// TwinCAT 3 PLC project PLC1
// ProgramVersion: 3.1.4026.16
// CompilerDefines: VISU_USEPROPERTYINFO
// libraries:
//   SH_Light, * (StroemHansen)
//   Tc2_EnOcean, * (Beckhoff Automation GmbH)
//   Tc2_Standard, * (Beckhoff Automation GmbH)
//   Tc2_System, * (Beckhoff Automation GmbH)
//   Tc2_Utilities, * (Beckhoff Automation GmbH)
//   Tc3_DALI, * (Beckhoff Automation GmbH)
//   Tc3_System_DK, * (Beckhoff - DK)
//   VisuDialogs, * (System)
// project tree:
//   DUTs/DALI/ E_DALIExtendedFadeTime.TcTLEO (not stored), ST_DALI102Parameters.TcDUT (not stored), ST_DALI103Parameters.TcDUT (not stored), ST_DALIMemoryBank.TcDUT (not stored), ST_DALI_GrpAssignment.TcDUT (not stored), ST_GroupSort.TcDUT (not stored)
//   DUTs/EnOcean/ ST_ReadSAB05.TcDUT (not stored), ST_WriteSAB05.TcDUT (not stored)
//   / FastTask.TcTTO (not stored), GlobalTextList.TcGTLO (not stored), PlcTask.TcTTO (not stored), Visualization Manager.TcVMO (not stored)
//   GVLs/ GVL_AHDataModbus.TcGVL, GVL_EnOcean.TcGVL, GVL_Skalering.TcGVL (not stored)
//   POUs/01_System/01_System/GVLs/ GVL_EtherCAT.TcGVL (not stored)
//   POUs/01_System/01_System/ P_SystemDK.TcPOU (not stored)
//   POUs/AHModbusComm/ P_AHModbusComm.TcPOU
//   POUs/Alle_Rum/Gange/Gang_1_212A/ P_Gang_1_212A.TcPOU, Visualization_4_307_1_1_1_1.TcVIS (excluded from build)
//   POUs/Alle_Rum/Gange/Gang_1_216/ P_Gang_1_216.TcPOU, Visualization_4_308_1_2_1.TcVIS (excluded from build)
//   POUs/Alle_Rum/Gange/Gang_6_210/ P_Gang_6_210.TcPOU, Visualization_4_308_1_2_1_1.TcVIS (excluded from build)
//   POUs/Alle_Rum/Rum_Med_DALI_Pir/Rum_1_213/ P_Rum_1_213.TcPOU, Visualization_5_356_2_1_1_1.TcVIS (excluded from build)
//   POUs/Alle_Rum/Rum_Med_DALI_Pir/Rum_6_235/ P_Rum_6_235.TcPOU, Visualization_5_356_2_1_1_1_1.TcVIS (excluded from build)
//   POUs/Alle_Rum/Rum_Med_DALI_Pir/Rum_1_215/ P_Rum_1_215.TcPOU, Visualization_4_307_1_1_3_1_1_1.TcVIS (excluded from build)
//   POUs/Alle_Rum/Rum_Med_DALI_Pir/Rum_1_217/ P_Rum_1_217.TcPOU, Visualization_5_356_2_1_1_2.TcVIS (excluded from build)
//   POUs/Alle_Rum/Rum_Med_DALI_Pir/Rum_1_219/ P_Rum_1_219.TcPOU, Visualization_5_356_2_1_1_3.TcVIS (excluded from build)
//   POUs/Alle_Rum/Rum_Med_DALI_Pir/Rum_6_226B/ P_Rum_6_226B.TcPOU, Visualization_5_356_2_1_1_3_1.TcVIS (excluded from build)
//   POUs/Alle_Rum/Rum_Med_DALI_Pir/Rum_1_220/ P_Rum_1_220.TcPOU, Visualization_5_356_2_1_1_4.TcVIS (excluded from build)
//   POUs/Alle_Rum/Rum_Med_DALI_Pir/Rum_1_222/ P_Rum_1_222.TcPOU, Visualization_5_356_2_1_1_5.TcVIS (excluded from build)
//   POUs/Alle_Rum/Rum_Med_DALI_Pir/Rum_1_223/ P_Rum_1_223.TcPOU, Visualization_5_356_2_1_1_6.TcVIS (excluded from build)
//   POUs/Alle_Rum/Rum_Med_DALI_Pir/Rum_1_218/ P_Rum_1_218.TcPOU, Visualization_5_356_2_1_1.TcVIS (excluded from build)
//   POUs/Alle_Rum/Rum_Med_DALI_Pir/Rum_6_223/ P_Rum_6_223.TcPOU, Visualization_5_356_2_1_1_6_1.TcVIS (excluded from build)
//   POUs/Alle_Rum/Rum_Med_DALI_Pir/Rum_6_225/ P_Rum_6_225.TcPOU, Visualization_5_356_2_1_1_6_1_10.TcVIS (excluded from build)
//   POUs/Alle_Rum/Rum_Med_DALI_Pir/Rum_6_224/ P_Rum_6_224.TcPOU, Visualization_5_356_2_1_1_6_1_1.TcVIS (excluded from build)
//   POUs/Alle_Rum/Rum_Med_DALI_Pir/Rum_6_226A/ P_Rum_6_226A.TcPOU, Visualization_5_356_2_1_1_6_1_2.TcVIS (excluded from build)
//   POUs/Alle_Rum/Rum_Med_DALI_Pir/Rum_6_227/ P_Rum_6_227.TcPOU, Visualization_5_356_2_1_1_6_1_3.TcVIS (excluded from build)
//   POUs/Alle_Rum/Rum_Med_DALI_Pir/Rum_6_228/ P_Rum_6_228.TcPOU, Visualization_5_356_2_1_1_6_1_4.TcVIS (excluded from build)
//   POUs/Alle_Rum/Rum_Med_DALI_Pir/Rum_6_229/ P_Rum_6_229.TcPOU, Visualization_5_356_2_1_1_6_1_5.TcVIS (excluded from build)
//   POUs/Alle_Rum/Rum_Med_DALI_Pir/Rum_6_230/ P_Rum_6_230.TcPOU, Visualization_5_356_2_1_1_6_1_6.TcVIS (excluded from build)
//   POUs/Alle_Rum/Rum_Med_DALI_Pir/Rum_6_231/ P_Rum_6_231.TcPOU, Visualization_5_356_2_1_1_6_1_7.TcVIS (excluded from build)
//   POUs/Alle_Rum/Rum_Med_DALI_Pir/Rum_6_233/ P_Rum_6_233.TcPOU, Visualization_5_356_2_1_1_6_1_8.TcVIS (excluded from build)
//   POUs/Alle_Rum/Trapper/ P_Trappe.TcPOU (excluded from build)
//   POUs/DALI/DALI_Setup/ DALI_Commissioning.TcPOU (not stored)
//   POUs/DALI/DALI_Setup/FBs/ FB_Part102Addressing.TcPOU (not stored), FB_Part102Commands.TcPOU (not stored), FB_Part102Groups.TcPOU, FB_Part102MemoryPages.TcPOU (not stored), FB_Part102Parameters.TcPOU (not stored), FB_Part102Scenes.TcPOU (not stored), FB_Part102SetFading.TcPOU (not stored), FB_Part103Addressing.TcPOU (not stored), FB_Part103Identify.TcPOU (not stored), FB_Part103MemoryPages.TcPOU (not stored), FB_Part103Parameters.TcPOU (not stored), FB_Part202Emergency.TcPOU (not stored), FB_Part205Incandescent.TcPOU, FB_Part207LED.TcPOU, FB_Part208Switching.TcPOU (not stored), FB_Part300GenericDevice.TcPOU (not stored), FB_Part301PushButton.TcPOU (not stored), FB_Part302AbsoluteInputDevice.TcPOU (not stored), FB_Part303OccupancySensor.TcPOU (not stored), FB_Part304LightSensor.TcPOU (not stored), GearType.TcPOU (not stored)
//   POUs/DALI/DALI_Setup/GVLs/ GVL_Internal.TcGVL (not stored)
//   POUs/DALI/DALI_Setup/VISUs/TextLists/ CommandOnTerminalEvent.TcTLO, DimmingCurve.TcTLO (not stored), EventPriority.TcTLO (not stored), EventScheme.TcTLO, ExtendedFadeTime.TcTLO, FadeRate.TcTLO (not stored), FadeTime.TcTLO (not stored), FastFadeTime.TcTLO (not stored), TextList_Dialogs.TcTLO (not stored)
//   POUs/DALI/DALI_Setup/VISUs/ Visu_DALICommissioning.TcVIS
//   POUs/DALI/DALI_Setup/VISUs/Visu_DALICommissioning/ Visu_KL6821Configuration.TcVIS (not stored) (excluded from build), Visu_Part102Addressing.TcVIS, Visu_Part102Commands.TcVIS (not stored), Visu_Part102Groups.TcVIS (not stored), Visu_Part102MemoryBank.TcVIS (not stored), Visu_Part102Parameters.TcVIS, Visu_Part102Scenes.TcVIS, Visu_Part102SetFading.TcVIS (not stored), Visu_Part103Addressing.TcVIS (not stored), Visu_Part103Identify.TcVIS (not stored), Visu_Part103MemoryBank.TcVIS (not stored), Visu_Part103Parameters.TcVIS, Visu_Part202.TcVIS (not stored), Visu_Part202Commands.TcVIS, Visu_Part202Parameters.TcVIS, Visu_Part202Status.TcVIS (not stored), Visu_Part205.TcVIS (not stored), Visu_Part205Parameters.TcVIS (not stored), Visu_Part205Status.TcVIS (not stored), Visu_Part207.TcVIS (not stored), Visu_Part207Parameters.TcVIS (not stored), Visu_Part207Status.TcVIS (not stored), Visu_Part208Switching.TcVIS (not stored), Visu_Part300GenericDevice.TcVIS (not stored), Visu_Part301PushButton.TcVIS (not stored), Visu_Part302AbsoluteInputDevice.TcVIS (not stored), Visu_Part303OccupancySensor.TcVIS (not stored), Visu_Part304LightSensor.TcVIS (not stored), Visu_Welcome.TcVIS (not stored)
//   POUs/DALI/PRGs/Background/ P_DALI_Background.TcPOU (not stored)
//   POUs/DALI/PRGs/Diag/ P_DALI_DIAG.TcPOU (not stored)
//   POUs/DALI/PRGs/EnergyData/ P_DALI_Energy_Firmware_Test.TcPOU (not stored) (excluded from build), P_DALI_Energy_Line.TcPOU (not stored)
//   POUs/EnOcean/ P_EnOcean.TcPOU
//   POUs/ MAIN.TcPOU
// real-time tasks:
//   TASK PlcTask: cycle T#40ms, priority 21, ADS port 350
//   TASK FastTask: cycle T#4ms, priority 20, ADS port 351
// I/O:
//   DEVICE Device 1 (Beckhoff CCAT)
//   DEVICE Device 3 (CX-BK)
//     Box 1 (CX-BK)
// variable links:
//   PLC1/PLC1 Instance <-> Device 3 (CX-BK)/Box 1 (CX-BK)
//     FastTask Inputs/P_DALI_Background.arrKL6821InData[1] @bit 16 <-> Term 3 (KL6821)/Channel 1/Data In 0
//     FastTask Inputs/P_DALI_Background.arrKL6821InData[1] @bit 24 <-> Term 3 (KL6821)/Channel 1/Data In 1
//     FastTask Inputs/P_DALI_Background.arrKL6821InData[1] @bit 32 <-> Term 3 (KL6821)/Channel 1/Data In 2
//     FastTask Inputs/P_DALI_Background.arrKL6821InData[1] @bit 40 <-> Term 3 (KL6821)/Channel 1/Data In 3
//     FastTask Inputs/P_DALI_Background.arrKL6821InData[2] @bit 16 <-> Term 4 (KL6821)/Channel 1/Data In 0
//     FastTask Inputs/P_DALI_Background.arrKL6821InData[2] @bit 24 <-> Term 4 (KL6821)/Channel 1/Data In 1
//     FastTask Inputs/P_DALI_Background.arrKL6821InData[2] @bit 32 <-> Term 4 (KL6821)/Channel 1/Data In 2
//     FastTask Inputs/P_DALI_Background.arrKL6821InData[2] @bit 40 <-> Term 4 (KL6821)/Channel 1/Data In 3
//     FastTask Inputs/P_DALI_Background.arrKL6821InData[3] @bit 16 <-> Term 5 (KL6821)/Channel 1/Data In 0
//     FastTask Inputs/P_DALI_Background.arrKL6821InData[3] @bit 24 <-> Term 5 (KL6821)/Channel 1/Data In 1
//     FastTask Inputs/P_DALI_Background.arrKL6821InData[3] @bit 32 <-> Term 5 (KL6821)/Channel 1/Data In 2
//     FastTask Inputs/P_DALI_Background.arrKL6821InData[3] @bit 40 <-> Term 5 (KL6821)/Channel 1/Data In 3
//     FastTask Inputs/P_DALI_Background.arrKL6821InData[4] @bit 16 <-> Term 6 (KL6821)/Channel 1/Data In 0
//     FastTask Inputs/P_DALI_Background.arrKL6821InData[4] @bit 24 <-> Term 6 (KL6821)/Channel 1/Data In 1
//     FastTask Inputs/P_DALI_Background.arrKL6821InData[4] @bit 32 <-> Term 6 (KL6821)/Channel 1/Data In 2
//     FastTask Inputs/P_DALI_Background.arrKL6821InData[4] @bit 40 <-> Term 6 (KL6821)/Channel 1/Data In 3
//     FastTask Inputs/P_DALI_Background.arrKL6821InData[{1..4}] <-> Term {3..6} (KL6821)/Channel 1/State  (4 links)
//     FastTask Inputs/P_EnOcean.stKL6581_in @bit 8 <-> Term 2 (KL6581)/Channel 1/Input CNODE
//     FastTask Inputs/P_EnOcean.stKL6581_in @bit {24..48 step 8} <-> Term 2 (KL6581)/Channel 1/Input DB{0..3}  (4 links)
//     FastTask Inputs/P_EnOcean.stKL6581_in @bit {56..80 step 8} <-> Term 2 (KL6581)/Channel 1/Input ID{0..3}  (4 links)
//     FastTask Inputs/P_EnOcean.stKL6581_in @bit 16 <-> Term 2 (KL6581)/Channel 1/Input ORG
//     FastTask Inputs/P_EnOcean.stKL6581_in @bit 88 <-> Term 2 (KL6581)/Channel 1/Input STATUS
//     FastTask Inputs/P_EnOcean.stKL6581_in <-> Term 2 (KL6581)/Channel 1/Status
//     FastTask Outputs/P_DALI_Background.arrKL6821OutData[{1..4}] <-> Term {3..6} (KL6821)/Channel 1/Ctrl  (4 links)
//     FastTask Outputs/P_DALI_Background.arrKL6821OutData[1] @bit 16 <-> Term 3 (KL6821)/Channel 1/Data Out 0
//     FastTask Outputs/P_DALI_Background.arrKL6821OutData[1] @bit 24 <-> Term 3 (KL6821)/Channel 1/Data Out 1
//     FastTask Outputs/P_DALI_Background.arrKL6821OutData[1] @bit 32 <-> Term 3 (KL6821)/Channel 1/Data Out 2
//     FastTask Outputs/P_DALI_Background.arrKL6821OutData[1] @bit 40 <-> Term 3 (KL6821)/Channel 1/Data Out 3
//     FastTask Outputs/P_DALI_Background.arrKL6821OutData[2] @bit 16 <-> Term 4 (KL6821)/Channel 1/Data Out 0
//     FastTask Outputs/P_DALI_Background.arrKL6821OutData[2] @bit 24 <-> Term 4 (KL6821)/Channel 1/Data Out 1
//     FastTask Outputs/P_DALI_Background.arrKL6821OutData[2] @bit 32 <-> Term 4 (KL6821)/Channel 1/Data Out 2
//     FastTask Outputs/P_DALI_Background.arrKL6821OutData[2] @bit 40 <-> Term 4 (KL6821)/Channel 1/Data Out 3
//     FastTask Outputs/P_DALI_Background.arrKL6821OutData[3] @bit 16 <-> Term 5 (KL6821)/Channel 1/Data Out 0
//     FastTask Outputs/P_DALI_Background.arrKL6821OutData[3] @bit 24 <-> Term 5 (KL6821)/Channel 1/Data Out 1
//     FastTask Outputs/P_DALI_Background.arrKL6821OutData[3] @bit 32 <-> Term 5 (KL6821)/Channel 1/Data Out 2
//     FastTask Outputs/P_DALI_Background.arrKL6821OutData[3] @bit 40 <-> Term 5 (KL6821)/Channel 1/Data Out 3
//     FastTask Outputs/P_DALI_Background.arrKL6821OutData[4] @bit 16 <-> Term 6 (KL6821)/Channel 1/Data Out 0
//     FastTask Outputs/P_DALI_Background.arrKL6821OutData[4] @bit 24 <-> Term 6 (KL6821)/Channel 1/Data Out 1
//     FastTask Outputs/P_DALI_Background.arrKL6821OutData[4] @bit 32 <-> Term 6 (KL6821)/Channel 1/Data Out 2
//     FastTask Outputs/P_DALI_Background.arrKL6821OutData[4] @bit 40 <-> Term 6 (KL6821)/Channel 1/Data Out 3
//     FastTask Outputs/P_EnOcean.stKL6581_out <-> Term 2 (KL6581)/Channel 1/Control
//     FastTask Outputs/P_EnOcean.stKL6581_out @bit 8 <-> Term 2 (KL6581)/Channel 1/Output CNODE
//     FastTask Outputs/P_EnOcean.stKL6581_out @bit {24..48 step 8} <-> Term 2 (KL6581)/Channel 1/Output DB{0..3}  (4 links)
//     FastTask Outputs/P_EnOcean.stKL6581_out @bit {56..80 step 8} <-> Term 2 (KL6581)/Channel 1/Output ID{0..3}  (4 links)
//     FastTask Outputs/P_EnOcean.stKL6581_out @bit 16 <-> Term 2 (KL6581)/Channel 1/Output ORG
//     FastTask Outputs/P_EnOcean.stKL6581_out @bit 88 <-> Term 2 (KL6581)/Channel 1/Output STATUS
//     PlcTask Inputs/MAIN.nCX8200_State <-> Inputs/State

// ---- GVLs/GVL_AHDataModbus.TcGVL
{attribute 'qualified_only'}
{attribute 'qualified_only'}
VAR_GLOBAL
//AH pir data out
	nAH_NeighborRoomsPir_Out		AT %MB600	: UINT;
	
//AH pir data in
	arrAH_NeighborRoomsPir_In								: ARRAY[1..byNumberOfAH_Neighbors] OF UINT;
	arrAH_NeighborRoomsPir										: ARRAY[1..byNumberOfAH_Neighbors] OF ARRAY[0..15] OF BOOL;
	
//Schneider data out
	nCX8200_State_MB						AT %MB1000		: UINT;
	arrFB_DALIDiagErrorId		(*AT %MW1002*)		: ARRAY[1..SH_Light.DALI_Param.MAX_DALIV2_LINES] OF UDINT;
	arrKL6821InDataStatus					AT %MB1014		: ARRAY[1..SH_Light.DALI_Param.MAX_DALIV2_LINES] OF WORD;
	arrDALILineShrtAddrErr				AT %MB1026		: ARRAY[1..SH_Light.DALI_Param.MAX_DALIV2_LINES] OF UINT;
	EnOceanError								AT %MB1038		: UINT;
	nTotalEnergy10kWh						AT %MB1040		: UINT;
	nMaxControlGearOperatingHours	AT %MB1042		: UINT;
	uiPirOffDelayTimeAllRooms_MB   AT %MB1044   : UINT := 30;
END_VAR

VAR_GLOBAL CONSTANT
	byNumberOfAH_Neighbors									: BYTE := 25;
END_VAR


(*
AH2-2 pirsignaler = arrAH_NeighborRoomsPir[1]
	---------- KOPI fra A_AHNeighborRoomsPirOut i AH2-2 ----------
	GVL_AHDataModbus.nAH_NeighborRoomsPir_Out.0		:= P_Gang_2_244A.bPirActive_MB;
	GVL_AHDataModbus.nAH_NeighborRoomsPir_Out.1		:= P_Gang_7_201.bPirActive_MB;
*)

(*
AH6-2 pirsignaler = arrAH_NeighborRoomsPir[2]
	---------- KOPI fra A_AHNeighborRoomsPirOut i AH6-2 ----------
	
*)

// ---- GVLs/GVL_EnOcean.TcGVL
{attribute 'qualified_only'}
VAR_GLOBAL

//Gange
	strEnOceanSwitch_Gang_1_216_Pendler     			: Tc2_EnOcean.STR_EnOceanSwitch;

//Rum
	strEnOceanSwitch_Rum_1_213_Indgang				: Tc2_EnOcean.STR_EnOceanSwitch;
	strEnOceanSwitch_Rum_1_213_Ekstra					: Tc2_EnOcean.STR_EnOceanSwitch;
	
	strEnOceanSwitch_Rum_1_215								: Tc2_EnOcean.STR_EnOceanSwitch;
	strEnOceanSwitch_Rum_1_217								: Tc2_EnOcean.STR_EnOceanSwitch;
	strEnOceanSwitch_Rum_1_218								: Tc2_EnOcean.STR_EnOceanSwitch;
	strEnOceanSwitch_Rum_1_219								: Tc2_EnOcean.STR_EnOceanSwitch;
	strEnOceanSwitch_Rum_1_220								: Tc2_EnOcean.STR_EnOceanSwitch;
	strEnOceanSwitch_Rum_1_222								: Tc2_EnOcean.STR_EnOceanSwitch;
	strEnOceanSwitch_Rum_1_223								: Tc2_EnOcean.STR_EnOceanSwitch;
	
	strEnOceanSwitch_Rum_6_223								: Tc2_EnOcean.STR_EnOceanSwitch;
	strEnOceanSwitch_Rum_6_224								: Tc2_EnOcean.STR_EnOceanSwitch;
	strEnOceanSwitch_Rum_6_225								: Tc2_EnOcean.STR_EnOceanSwitch;
	strEnOceanSwitch_Rum_6_226A							: Tc2_EnOcean.STR_EnOceanSwitch;
	
	strEnOceanSwitch_Rum_6_226B_Indgang				: Tc2_EnOcean.STR_EnOceanSwitch;
	strEnOceanSwitch_Rum_6_226B_Pendler				: Tc2_EnOcean.STR_EnOceanSwitch;
	
	strEnOceanSwitch_Rum_6_227								: Tc2_EnOcean.STR_EnOceanSwitch;
	strEnOceanSwitch_Rum_6_228								: Tc2_EnOcean.STR_EnOceanSwitch;
	strEnOceanSwitch_Rum_6_229								: Tc2_EnOcean.STR_EnOceanSwitch;
	strEnOceanSwitch_Rum_6_230								: Tc2_EnOcean.STR_EnOceanSwitch;
	strEnOceanSwitch_Rum_6_231								: Tc2_EnOcean.STR_EnOceanSwitch;
	strEnOceanSwitch_Rum_6_233								: Tc2_EnOcean.STR_EnOceanSwitch;
	
	strEnOceanSwitch_Rum_6_235_Indgang				: Tc2_EnOcean.STR_EnOceanSwitch;
	strEnOceanSwitch_Rum_6_235_Ekstra					: Tc2_EnOcean.STR_EnOceanSwitch;
END_VAR

// ---- POUs/AHModbusComm/P_AHModbusComm.TcPOU
PROGRAM P_AHModbusComm
VAR
	arrfbReadAHPirData	: ARRAY[1..GVL_AHDataModbus.byNumberOfAH_Neighbors] OF SH_Light.FB_ReadAHPirData;
	arrReadAHPirData		: ARRAY[1..GVL_AHDataModbus.byNumberOfAH_Neighbors] OF BOOL;
	
	arrfbTriggerPulses			: ARRAY[1..GVL_AHDataModbus.byNumberOfAH_Neighbors] OF SH_Light.FB_ClockPulse;
	arrGeneratePulses			: ARRAY[1..GVL_AHDataModbus.byNumberOfAH_Neighbors] OF BOOL := [GVL_AHDataModbus.byNumberOfAH_Neighbors(TRUE)];
	tTimeInterval					: TIME := T#1S;
	tPulseTime					: TIME := T#1S;
	
	byLineId						: BYTE;
	byAHId						: BYTE;
	
		
	fbWritePirDelayTime		: R_TRIG;
	bRunOverrideOnce		: BOOL := FALSE;
	bEnableDelayTimeOverride : BOOL := FALSE;
	uiPirOffDelayTimeAllRooms : UINT := 30;
END_VAR

VAR CONSTANT
	arrnMBAddr					: ARRAY[1..GVL_AHDataModbus.byNumberOfAH_Neighbors] OF WORD := [GVL_AHDataModbus.byNumberOfAH_Neighbors(12588)]; //modbus-adresser (%MB600=>12588 default)
	arrstNeighborIPAddr		: ARRAY[1..GVL_AHDataModbus.byNumberOfAH_Neighbors] OF SH_Light.ST_NeighborIP := [
																						(sPLCName := 'AH1-1', sIP := '172.24.195.161', IsNeighbor := FALSE),
																						(sPLCName := 'AH1-2', sIP := '172.24.195.162', IsNeighbor := FALSE),	//Local must be false
																						(sPLCName := 'AH1-3', sIP := '172.24.195.163', IsNeighbor := FALSE),
																						(sPLCName := 'AH2-1', sIP := '172.24.195.164', IsNeighbor := FALSE),
																					(sPLCName := 'AH2-2', sIP := '172.24.195.165', IsNeighbor := TRUE),
																						(sPLCName := 'AH2-3', sIP := '172.24.195.166', IsNeighbor := FALSE),
																						(sPLCName := 'AH2-4', sIP := '172.24.195.167', IsNeighbor := FALSE),
																						(sPLCName := 'AH2-5', sIP := '172.24.195.168', IsNeighbor := FALSE),
																						(sPLCName := 'AH3-2', sIP := '172.24.195.169', IsNeighbor := FALSE),
																						(sPLCName := 'AH3-3', sIP := '172.24.195.170', IsNeighbor := FALSE),
																						(sPLCName := 'AH3-4', sIP := '172.24.195.171', IsNeighbor := FALSE),
																						(sPLCName := 'AH3-5', sIP := '172.24.195.172', IsNeighbor := FALSE),
																						(sPLCName := 'AH4-1', sIP := '172.24.195.173', IsNeighbor := FALSE),
																						(sPLCName := 'AH4-2', sIP := '172.24.195.174', IsNeighbor := FALSE),
																						(sPLCName := 'AH4-3', sIP := '172.24.195.175', IsNeighbor := FALSE),
																						(sPLCName := 'AH4-4', sIP := '172.24.195.176', IsNeighbor := FALSE),
																						(sPLCName := 'AH4-5', sIP := '172.24.195.177', IsNeighbor := FALSE),
																						(sPLCName := 'AH5-1', sIP := '172.24.195.178', IsNeighbor := FALSE),
																						(sPLCName := 'AH5-2', sIP := '172.24.195.179', IsNeighbor := FALSE),
																						(sPLCName := 'AH5-3', sIP := '172.24.195.180', IsNeighbor := FALSE),
																						(sPLCName := 'AH5-4', sIP := '172.24.195.181', IsNeighbor := FALSE),
																						(sPLCName := 'AH5-5', sIP := '172.24.195.182', IsNeighbor := FALSE),
																						(sPLCName := 'AH6-1', sIP := '172.24.195.183', IsNeighbor := FALSE),
																					(sPLCName := 'AH6-2', sIP := '172.24.195.184', IsNeighbor := TRUE),
																						(sPLCName := 'AH6-3', sIP := '172.24.195.185', IsNeighbor := FALSE)];
																					//	(sPLCName := 'AH3-1', sIP := '172.24.195.186', IsNeighbor := TRUE) //when ready
END_VAR

A_AHNeighborRoomsPirIn();
A_AHNeighborRoomsPirOut();
A_DALILineShrtAddrErr();
A_DelayTimeAllRooms();

ACTION A_AHNeighborRoomsPirIn:
FOR byAHId := 1 TO GVL_AHDataModbus.byNumberOfAH_Neighbors DO
	IF arrstNeighborIPAddr[byAHId].IsNeighbor THEN
		//Generate Pulses
		arrfbTriggerPulses[byAHId](bGenerateClockPulses:= arrGeneratePulses[byAHId], tTimeInterval:= tTimeInterval, tPulseTime:= tPulseTime);
		arrReadAHPirData[byAHId]:= arrfbTriggerPulses[byAHId].bPulse;
		//Read data
		arrfbReadAHPirData[byAHId](	bReadAHPirData				:=	arrReadAHPirData[byAHId],
														sIPAddr							:=	arrstNeighborIPAddr[byAHId].sIP,
														nMBAddr							:=	arrnMBAddr[byAHId],
														nMBDataBuffer				:=	GVL_AHDataModbus.arrAH_NeighborRoomsPir_In[byAHId],
														arrAH_NeighborRoomsPir	=>GVL_AHDataModbus.arrAH_NeighborRoomsPir[byAHId]);
	END_IF
END_FOR
END_ACTION

ACTION A_AHNeighborRoomsPirOut:
GVL_AHDataModbus.nAH_NeighborRoomsPir_Out.0 := P_Gang_1_216.bPirActive_MB;
GVL_AHDataModbus.nAH_NeighborRoomsPir_Out.1 := P_Gang_6_210.bPirActive_MB;
//GVL_AHDataModbus.nAH_NeighborRoomsPir_Out.2 :=
//GVL_AHDataModbus.nAH_NeighborRoomsPir_Out.3 := 
//GVL_AHDataModbus.nAH_NeighborRoomsPir_Out.4 :=
//GVL_AHDataModbus.nAH_NeighborRoomsPir_Out.5 := 
//GVL_AHDataModbus.nAH_NeighborRoomsPir_Out.6 :=
//GVL_AHDataModbus.nAH_NeighborRoomsPir_Out.7 := 
//GVL_AHDataModbus.nAH_NeighborRoomsPir_Out.8 :=
//GVL_AHDataModbus.nAH_NeighborRoomsPir_Out.9 := 
//GVL_AHDataModbus.nAH_NeighborRoomsPir_Out.10 :=
//GVL_AHDataModbus.nAH_NeighborRoomsPir_Out.11 := 
//GVL_AHDataModbus.nAH_NeighborRoomsPir_Out.12 := 
//GVL_AHDataModbus.nAH_NeighborRoomsPir_Out.13 := 
//GVL_AHDataModbus.nAH_NeighborRoomsPir_Out.14 := 
//GVL_AHDataModbus.nAH_NeighborRoomsPir_Out.15 :=
END_ACTION

ACTION A_DALILineShrtAddrErr:
FOR  byLineId := 1 TO SH_Light.DALI_Param.MAX_DALIV2_LINES DO
	GVL_AHDataModbus.arrDALILineShrtAddrErr[byLineId] :=  TO_UINT(SH_Light.GVL_DALI_LatestError.arrLineShrtAddr[byLineId]);
END_FOR
END_ACTION

ACTION A_DelayTimeAllRooms:

fbWritePirDelayTime(CLK := GVL_AHDataModbus.uiPirOffDelayTimeAllRooms_MB<>uiPirOffDelayTimeAllRooms);

IF fbWritePirDelayTime.Q THEN
	bRunOverrideOnce := TRUE;
	bEnableDelayTimeOverride := TRUE;
	
//Indsæt kode
P_Gang_1_212A.fbWritePirDelayTIme(bEnableOverride := bEnableDelayTimeOverride, nOverRideValue := GVL_AHDataModbus.uiPirOffDelayTimeAllRooms_MB, nValIn1 := GVL_AHDataModbus.uiPirOffDelayTimeAllRooms_MB, nValIn2 := uiPirOffDelayTimeAllRooms);
P_Gang_1_216.fbWritePirDelayTIme(bEnableOverride := bEnableDelayTimeOverride, nOverRideValue := GVL_AHDataModbus.uiPirOffDelayTimeAllRooms_MB, nValIn1 := GVL_AHDataModbus.uiPirOffDelayTimeAllRooms_MB, nValIn2 := uiPirOffDelayTimeAllRooms);
P_Gang_6_210.fbWritePirDelayTIme(bEnableOverride := bEnableDelayTimeOverride, nOverRideValue := GVL_AHDataModbus.uiPirOffDelayTimeAllRooms_MB, nValIn1 := GVL_AHDataModbus.uiPirOffDelayTimeAllRooms_MB, nValIn2 := uiPirOffDelayTimeAllRooms);
P_Rum_1_213.fbWritePirDelayTIme(bEnableOverride := bEnableDelayTimeOverride, nOverRideValue := GVL_AHDataModbus.uiPirOffDelayTimeAllRooms_MB, nValIn1 := GVL_AHDataModbus.uiPirOffDelayTimeAllRooms_MB, nValIn2 := uiPirOffDelayTimeAllRooms);
P_Rum_1_215.fbWritePirDelayTIme(bEnableOverride := bEnableDelayTimeOverride, nOverRideValue := GVL_AHDataModbus.uiPirOffDelayTimeAllRooms_MB, nValIn1 := GVL_AHDataModbus.uiPirOffDelayTimeAllRooms_MB, nValIn2 := uiPirOffDelayTimeAllRooms);
P_Rum_1_217.fbWritePirDelayTIme(bEnableOverride := bEnableDelayTimeOverride, nOverRideValue := GVL_AHDataModbus.uiPirOffDelayTimeAllRooms_MB, nValIn1 := GVL_AHDataModbus.uiPirOffDelayTimeAllRooms_MB, nValIn2 := uiPirOffDelayTimeAllRooms);
P_Rum_1_218.fbWritePirDelayTIme(bEnableOverride := bEnableDelayTimeOverride, nOverRideValue := GVL_AHDataModbus.uiPirOffDelayTimeAllRooms_MB, nValIn1 := GVL_AHDataModbus.uiPirOffDelayTimeAllRooms_MB, nValIn2 := uiPirOffDelayTimeAllRooms);
P_Rum_1_219.fbWritePirDelayTIme(bEnableOverride := bEnableDelayTimeOverride, nOverRideValue := GVL_AHDataModbus.uiPirOffDelayTimeAllRooms_MB, nValIn1 := GVL_AHDataModbus.uiPirOffDelayTimeAllRooms_MB, nValIn2 := uiPirOffDelayTimeAllRooms);
P_Rum_1_222.fbWritePirDelayTIme(bEnableOverride := bEnableDelayTimeOverride, nOverRideValue := GVL_AHDataModbus.uiPirOffDelayTimeAllRooms_MB, nValIn1 := GVL_AHDataModbus.uiPirOffDelayTimeAllRooms_MB, nValIn2 := uiPirOffDelayTimeAllRooms);
P_Rum_1_220.fbWritePirDelayTIme(bEnableOverride := bEnableDelayTimeOverride, nOverRideValue := GVL_AHDataModbus.uiPirOffDelayTimeAllRooms_MB, nValIn1 := GVL_AHDataModbus.uiPirOffDelayTimeAllRooms_MB, nValIn2 := uiPirOffDelayTimeAllRooms);
P_Rum_1_223.fbWritePirDelayTIme(bEnableOverride := bEnableDelayTimeOverride, nOverRideValue := GVL_AHDataModbus.uiPirOffDelayTimeAllRooms_MB, nValIn1 := GVL_AHDataModbus.uiPirOffDelayTimeAllRooms_MB, nValIn2 := uiPirOffDelayTimeAllRooms);
P_Rum_6_223.fbWritePirDelayTIme(bEnableOverride := bEnableDelayTimeOverride, nOverRideValue := GVL_AHDataModbus.uiPirOffDelayTimeAllRooms_MB, nValIn1 := GVL_AHDataModbus.uiPirOffDelayTimeAllRooms_MB, nValIn2 := uiPirOffDelayTimeAllRooms);
P_Rum_6_224.fbWritePirDelayTIme(bEnableOverride := bEnableDelayTimeOverride, nOverRideValue := GVL_AHDataModbus.uiPirOffDelayTimeAllRooms_MB, nValIn1 := GVL_AHDataModbus.uiPirOffDelayTimeAllRooms_MB, nValIn2 := uiPirOffDelayTimeAllRooms);
P_Rum_6_225.fbWritePirDelayTIme(bEnableOverride := bEnableDelayTimeOverride, nOverRideValue := GVL_AHDataModbus.uiPirOffDelayTimeAllRooms_MB, nValIn1 := GVL_AHDataModbus.uiPirOffDelayTimeAllRooms_MB, nValIn2 := uiPirOffDelayTimeAllRooms);
P_Rum_6_226A.fbWritePirDelayTIme(bEnableOverride := bEnableDelayTimeOverride, nOverRideValue := GVL_AHDataModbus.uiPirOffDelayTimeAllRooms_MB, nValIn1 := GVL_AHDataModbus.uiPirOffDelayTimeAllRooms_MB, nValIn2 := uiPirOffDelayTimeAllRooms);
P_Rum_6_226B.fbWritePirDelayTIme(bEnableOverride := bEnableDelayTimeOverride, nOverRideValue := GVL_AHDataModbus.uiPirOffDelayTimeAllRooms_MB, nValIn1 := GVL_AHDataModbus.uiPirOffDelayTimeAllRooms_MB, nValIn2 := uiPirOffDelayTimeAllRooms);
P_Rum_6_227.fbWritePirDelayTIme(bEnableOverride := bEnableDelayTimeOverride, nOverRideValue := GVL_AHDataModbus.uiPirOffDelayTimeAllRooms_MB, nValIn1 := GVL_AHDataModbus.uiPirOffDelayTimeAllRooms_MB, nValIn2 := uiPirOffDelayTimeAllRooms);
P_Rum_6_228.fbWritePirDelayTIme(bEnableOverride := bEnableDelayTimeOverride, nOverRideValue := GVL_AHDataModbus.uiPirOffDelayTimeAllRooms_MB, nValIn1 := GVL_AHDataModbus.uiPirOffDelayTimeAllRooms_MB, nValIn2 := uiPirOffDelayTimeAllRooms);
P_Rum_6_229.fbWritePirDelayTIme(bEnableOverride := bEnableDelayTimeOverride, nOverRideValue := GVL_AHDataModbus.uiPirOffDelayTimeAllRooms_MB, nValIn1 := GVL_AHDataModbus.uiPirOffDelayTimeAllRooms_MB, nValIn2 := uiPirOffDelayTimeAllRooms);
P_Rum_6_230.fbWritePirDelayTIme(bEnableOverride := bEnableDelayTimeOverride, nOverRideValue := GVL_AHDataModbus.uiPirOffDelayTimeAllRooms_MB, nValIn1 := GVL_AHDataModbus.uiPirOffDelayTimeAllRooms_MB, nValIn2 := uiPirOffDelayTimeAllRooms);
P_Rum_6_231.fbWritePirDelayTIme(bEnableOverride := bEnableDelayTimeOverride, nOverRideValue := GVL_AHDataModbus.uiPirOffDelayTimeAllRooms_MB, nValIn1 := GVL_AHDataModbus.uiPirOffDelayTimeAllRooms_MB, nValIn2 := uiPirOffDelayTimeAllRooms);
P_Rum_6_233.fbWritePirDelayTIme(bEnableOverride := bEnableDelayTimeOverride, nOverRideValue := GVL_AHDataModbus.uiPirOffDelayTimeAllRooms_MB, nValIn1 := GVL_AHDataModbus.uiPirOffDelayTimeAllRooms_MB, nValIn2 := uiPirOffDelayTimeAllRooms);
P_Rum_6_235.fbWritePirDelayTIme(bEnableOverride := bEnableDelayTimeOverride, nOverRideValue := GVL_AHDataModbus.uiPirOffDelayTimeAllRooms_MB, nValIn1 := GVL_AHDataModbus.uiPirOffDelayTimeAllRooms_MB, nValIn2 := uiPirOffDelayTimeAllRooms);

ELSE
	IF bRunOverrideOnce THEN
		bEnableDelayTimeOverride := FALSE;
		
		//Indsæt kode
P_Gang_1_212A.fbWritePirDelayTIme(bEnableOverride := bEnableDelayTimeOverride, nOverRideValue := GVL_AHDataModbus.uiPirOffDelayTimeAllRooms_MB, nValIn1 := GVL_AHDataModbus.uiPirOffDelayTimeAllRooms_MB, nValIn2 := uiPirOffDelayTimeAllRooms);
P_Gang_1_216.fbWritePirDelayTIme(bEnableOverride := bEnableDelayTimeOverride, nOverRideValue := GVL_AHDataModbus.uiPirOffDelayTimeAllRooms_MB, nValIn1 := GVL_AHDataModbus.uiPirOffDelayTimeAllRooms_MB, nValIn2 := uiPirOffDelayTimeAllRooms);
P_Gang_6_210.fbWritePirDelayTIme(bEnableOverride := bEnableDelayTimeOverride, nOverRideValue := GVL_AHDataModbus.uiPirOffDelayTimeAllRooms_MB, nValIn1 := GVL_AHDataModbus.uiPirOffDelayTimeAllRooms_MB, nValIn2 := uiPirOffDelayTimeAllRooms);
P_Rum_1_213.fbWritePirDelayTIme(bEnableOverride := bEnableDelayTimeOverride, nOverRideValue := GVL_AHDataModbus.uiPirOffDelayTimeAllRooms_MB, nValIn1 := GVL_AHDataModbus.uiPirOffDelayTimeAllRooms_MB, nValIn2 := uiPirOffDelayTimeAllRooms);
P_Rum_1_215.fbWritePirDelayTIme(bEnableOverride := bEnableDelayTimeOverride, nOverRideValue := GVL_AHDataModbus.uiPirOffDelayTimeAllRooms_MB, nValIn1 := GVL_AHDataModbus.uiPirOffDelayTimeAllRooms_MB, nValIn2 := uiPirOffDelayTimeAllRooms);
P_Rum_1_217.fbWritePirDelayTIme(bEnableOverride := bEnableDelayTimeOverride, nOverRideValue := GVL_AHDataModbus.uiPirOffDelayTimeAllRooms_MB, nValIn1 := GVL_AHDataModbus.uiPirOffDelayTimeAllRooms_MB, nValIn2 := uiPirOffDelayTimeAllRooms);
P_Rum_1_218.fbWritePirDelayTIme(bEnableOverride := bEnableDelayTimeOverride, nOverRideValue := GVL_AHDataModbus.uiPirOffDelayTimeAllRooms_MB, nValIn1 := GVL_AHDataModbus.uiPirOffDelayTimeAllRooms_MB, nValIn2 := uiPirOffDelayTimeAllRooms);
P_Rum_1_219.fbWritePirDelayTIme(bEnableOverride := bEnableDelayTimeOverride, nOverRideValue := GVL_AHDataModbus.uiPirOffDelayTimeAllRooms_MB, nValIn1 := GVL_AHDataModbus.uiPirOffDelayTimeAllRooms_MB, nValIn2 := uiPirOffDelayTimeAllRooms);
P_Rum_1_222.fbWritePirDelayTIme(bEnableOverride := bEnableDelayTimeOverride, nOverRideValue := GVL_AHDataModbus.uiPirOffDelayTimeAllRooms_MB, nValIn1 := GVL_AHDataModbus.uiPirOffDelayTimeAllRooms_MB, nValIn2 := uiPirOffDelayTimeAllRooms);
P_Rum_1_220.fbWritePirDelayTIme(bEnableOverride := bEnableDelayTimeOverride, nOverRideValue := GVL_AHDataModbus.uiPirOffDelayTimeAllRooms_MB, nValIn1 := GVL_AHDataModbus.uiPirOffDelayTimeAllRooms_MB, nValIn2 := uiPirOffDelayTimeAllRooms);
P_Rum_1_223.fbWritePirDelayTIme(bEnableOverride := bEnableDelayTimeOverride, nOverRideValue := GVL_AHDataModbus.uiPirOffDelayTimeAllRooms_MB, nValIn1 := GVL_AHDataModbus.uiPirOffDelayTimeAllRooms_MB, nValIn2 := uiPirOffDelayTimeAllRooms);
P_Rum_6_223.fbWritePirDelayTIme(bEnableOverride := bEnableDelayTimeOverride, nOverRideValue := GVL_AHDataModbus.uiPirOffDelayTimeAllRooms_MB, nValIn1 := GVL_AHDataModbus.uiPirOffDelayTimeAllRooms_MB, nValIn2 := uiPirOffDelayTimeAllRooms);
P_Rum_6_224.fbWritePirDelayTIme(bEnableOverride := bEnableDelayTimeOverride, nOverRideValue := GVL_AHDataModbus.uiPirOffDelayTimeAllRooms_MB, nValIn1 := GVL_AHDataModbus.uiPirOffDelayTimeAllRooms_MB, nValIn2 := uiPirOffDelayTimeAllRooms);
P_Rum_6_225.fbWritePirDelayTIme(bEnableOverride := bEnableDelayTimeOverride, nOverRideValue := GVL_AHDataModbus.uiPirOffDelayTimeAllRooms_MB, nValIn1 := GVL_AHDataModbus.uiPirOffDelayTimeAllRooms_MB, nValIn2 := uiPirOffDelayTimeAllRooms);
P_Rum_6_226A.fbWritePirDelayTIme(bEnableOverride := bEnableDelayTimeOverride, nOverRideValue := GVL_AHDataModbus.uiPirOffDelayTimeAllRooms_MB, nValIn1 := GVL_AHDataModbus.uiPirOffDelayTimeAllRooms_MB, nValIn2 := uiPirOffDelayTimeAllRooms);
P_Rum_6_226B.fbWritePirDelayTIme(bEnableOverride := bEnableDelayTimeOverride, nOverRideValue := GVL_AHDataModbus.uiPirOffDelayTimeAllRooms_MB, nValIn1 := GVL_AHDataModbus.uiPirOffDelayTimeAllRooms_MB, nValIn2 := uiPirOffDelayTimeAllRooms);
P_Rum_6_227.fbWritePirDelayTIme(bEnableOverride := bEnableDelayTimeOverride, nOverRideValue := GVL_AHDataModbus.uiPirOffDelayTimeAllRooms_MB, nValIn1 := GVL_AHDataModbus.uiPirOffDelayTimeAllRooms_MB, nValIn2 := uiPirOffDelayTimeAllRooms);
P_Rum_6_228.fbWritePirDelayTIme(bEnableOverride := bEnableDelayTimeOverride, nOverRideValue := GVL_AHDataModbus.uiPirOffDelayTimeAllRooms_MB, nValIn1 := GVL_AHDataModbus.uiPirOffDelayTimeAllRooms_MB, nValIn2 := uiPirOffDelayTimeAllRooms);
P_Rum_6_229.fbWritePirDelayTIme(bEnableOverride := bEnableDelayTimeOverride, nOverRideValue := GVL_AHDataModbus.uiPirOffDelayTimeAllRooms_MB, nValIn1 := GVL_AHDataModbus.uiPirOffDelayTimeAllRooms_MB, nValIn2 := uiPirOffDelayTimeAllRooms);
P_Rum_6_230.fbWritePirDelayTIme(bEnableOverride := bEnableDelayTimeOverride, nOverRideValue := GVL_AHDataModbus.uiPirOffDelayTimeAllRooms_MB, nValIn1 := GVL_AHDataModbus.uiPirOffDelayTimeAllRooms_MB, nValIn2 := uiPirOffDelayTimeAllRooms);
P_Rum_6_231.fbWritePirDelayTIme(bEnableOverride := bEnableDelayTimeOverride, nOverRideValue := GVL_AHDataModbus.uiPirOffDelayTimeAllRooms_MB, nValIn1 := GVL_AHDataModbus.uiPirOffDelayTimeAllRooms_MB, nValIn2 := uiPirOffDelayTimeAllRooms);
P_Rum_6_233.fbWritePirDelayTIme(bEnableOverride := bEnableDelayTimeOverride, nOverRideValue := GVL_AHDataModbus.uiPirOffDelayTimeAllRooms_MB, nValIn1 := GVL_AHDataModbus.uiPirOffDelayTimeAllRooms_MB, nValIn2 := uiPirOffDelayTimeAllRooms);
P_Rum_6_235.fbWritePirDelayTIme(bEnableOverride := bEnableDelayTimeOverride, nOverRideValue := GVL_AHDataModbus.uiPirOffDelayTimeAllRooms_MB, nValIn1 := GVL_AHDataModbus.uiPirOffDelayTimeAllRooms_MB, nValIn2 := uiPirOffDelayTimeAllRooms);

		bRunOverrideOnce := FALSE;
	END_IF
END_IF
END_ACTION

END_PROGRAM

// ---- POUs/Alle_Rum/Gange/Gang_1_216/P_Gang_1_216.TcPOU
PROGRAM P_Gang_1_216
(*
Gangen består af en lysgruppe og et ekstra armatur - L2G2 og L1S38 - på to forskellige linjer
både gruppe og ekstra armatur afhænger af samme PIR-input : pir-adr. 5, 6 og 10 på DALI-linje 2 og pir-adr. 4 på DALI-linje 4
Derfor oprettes to adskilte reguleringer med samme PV. Dvs., at knapfunktion og pirfunktion forbliver den samme.
Der oprettes to sensor setups, som samles i A_Sensor.
Gangen nabostyres af Gang_1_216 fra AH2-2 og udvalgte rum på gangen
*)
VAR
	arrfbLysGruppe			: ARRAY [1..2] OF FB_Light_Type_B;
	arrstDaliSetupGruppe	: ARRAY[1..2] OF SH_Light.ST_DALI_RoomSetup := 
	
													[(	byShrtAdr_Prim	:= 11, 
														byGrpAdr_Prim		:= 2, 
														eMod_Prim			:= E_DALIAddressType.Group, 
														//byShrtAdr_Sec		:= 1, 
														//byGrpAdr_Sec		:= 1, 
														//eMod_Sec			:= E_DALIAddressType.Short, 
														byShrtAdr_Supl		:= 26,
														//byGrpAdr_Supl := 1,
														eMod_Supl			:= E_DALIAddressType.Short,
														DALI_LINE_NUM_PRIM	:= arrDALI_LINE_NUM_LIGHT[1], 
														DALI_LINE_NUM_SEC		:= 0, //0 = ingen zonestyring/vinduerække
														DALI_LINE_NUM_SUPL	:= arrDALI_LINE_NUM_PENDANTS[1]),
														
													(	byShrtAdr_Prim	:= 38, 
														byGrpAdr_Prim		:= 1, 
														eMod_Prim			:= E_DALIAddressType.Short, 
														//byShrtAdr_Sec		:= 1, 
														//byGrpAdr_Sec		:= 1, 
														//eMod_Sec			:= E_DALIAddressType.Short, 
														//byShrtAdr_Supl		:= 1,
														//byGrpAdr_Supl := 1,
														//eMod_Supl			:= E_DALIAddressType.Short, 
														DALI_LINE_NUM_PRIM	:= arrDALI_LINE_NUM_LIGHT[2], 
														DALI_LINE_NUM_SEC		:= 0, 
														DALI_LINE_NUM_SUPL	:= arrDALI_LINE_NUM_PENDANTS[2])];
	
	arrstLiveDataGruppe			: ARRAY [1..2] OF SH_Light.ST_LiveData;
	arrRunTuningGruppe			: ARRAY[1..2] OF BOOL;
	
	bTopButtonZone1				: BOOL;
	bTopButtonZone1_Visu		: BOOL;
	bBottomButtonZone1			: BOOL;
	bBottomButtonZone1_Visu	: BOOL;
	bButtonZone2					: BOOL;
	bNeighborRoomsPir			: BOOL;
	fLuxOn								: REAL;
	fLuxDim							: REAL;
	tPIRDim							: TIME;
	tPIROff							: TIME;
	fOffsetSec						: REAL := 20;
	bOccupiedRoom				: BOOL;

// Sensor Settings
	fbSensor						: SH_Light.FB_NIKO_P46xx_3Pcs;
	arrSensorAddr				: ARRAY[1..3] OF BYTE :=[5,6,10];  
	bInitialize						: BOOL := TRUE;
	stDaliSensorSetup			: ST_DALI_NIKOP46SetupData;
	arrInitErr						: ARRAY [1..3] OF BOOL;
	arrInitDone					: ARRAY [1..3] OF BOOL;
	arrSensorScales				: ARRAY [1..10] OF SH_Light.ST_DALI_SensorScaleMode := [
																							(fMeassureMaxSensor := rMeassure_Zone10, fReadMaxSensor := rRead_Zone10),
																							(fMeassureMaxSensor := rMeassure_Zone10, fReadMaxSensor := rRead_Zone10),
																							(fMeassureMaxSensor := rMeassure_Zone10, fReadMaxSensor := rRead_Zone10),
																							7(())];
	
	//Setup af sensorer på forskellige linjer kan ikke håndteres med ARRAYS som sædvanlig, da der kun er 1 sensor på setup 2.
	fbSensor2						: SH_Light.FB_NIKO_P46xx_1Pcs;
	bySensor2Addr				: BYTE := 4;
	bInitialize2						: BOOL := TRUE;
	stDaliSensor2Setup		: ST_DALI_NIKOP46SetupData;
	bInitErr2						: BOOL;
	bInitDone2					: BOOL;
	arrSensor2Scales			: ARRAY [1..10] OF SH_Light.ST_DALI_SensorScaleMode := [
																							(fMeassureMaxSensor := 1023, fReadMaxSensor := 1023),
																							9(())];
																					
	bCancelHoldTimerOccupancy	: BOOL;
	
(*	eEventPriorityOccupancy		: E_DALIEventPriority := E_DALIEVENTPRIORITY.Middle;
	nHoldTimerOccupancy			: WORD := 5; // Value in s. 	
	nReportTimerOccupancy		: BYTE := 120; // Value in s, Preset manufacturer value
	nDeadtimeTimerOccupancy		: WORD := 100; // Value in ms, Predefined Value of DALI Standard
	bCancelHoldTimerOccupancy	: BOOL;
	nSensitivityOccupancy		: BYTE:= 3; //setting Sensivity (0..4) 0 (Off), 1 (Min), 2(Low), 3(High) and 4 (Max)

	bEnableLuxEvent				: BOOL;
	eEventPriorityBrightness	: E_DALIEventPriority := E_DALIEVENTPRIORITY.Middle;
	nDeadtimeTimerBrightness	: WORD := 1500; // Value in ms, Predefined Value of DALI Standard
	nHysteresisBrightness		: BYTE := 2; // Value in %
	nHysteresisMinBrightness	: BYTE := 10; // Absolute Value, depending on the manufacturer specific resolution
	nReportTimerBrightness		: BYTE := 120; // Value in s, Preset manufacturer value
*)

	//ModbusComm setup
	
	fbWriteSPLuxLevel				: SH_Light.FB_TwoVal_SelectOne_RTrigChange;
	fbWritePirDelayTIme			: SH_Light.FB_TwoVal_SelectOne_RTrigChange;
	stRoomDataPLC					: SH_Light.ST_RoomDataPLC	:=	(
																		uiPirOffDelayTime	:= 30,
																		uiSpLuxLevel			:= 500,
																		uiPirDimDelayTime	:= 15,
																		uiSpDimLuxLevel		:= 200);
																		
	fbBallastOnHours				: SH_Light.FB_CountOnHours;
	bEnableHourCount			: BOOL := TRUE;
	
	//Non-persistent modbus data
	bPirActive_MB					AT %MX32.0	: BOOL;				//bPirLys i gammel kode
	uiActLuxLevel_MB			AT %MB36		: UINT;				//intHMIAktueltLux i gammel kode
	uiActLightLevelPct_MB	AT %MB40		: UINT;				//intDALI_Gruppe1_Lysniveau i gammel kode
	
	//For Conversion
	uiPirOffMinutes						: UINT;
	udTimeScaling						: UDINT := 60000;
	uiLuxOn								: UINT;
	
	//max values checks
	uiMaxLuxLevel						: UINT := 1023;
	uiMaxPirOffMinutes				: UINT := 180;

END_VAR

VAR CONSTANT
	Sensor_DALI_LINE_NUM		: BYTE := 2;
	Sensor2_DALI_LINE_NUM	: BYTE := 4;
    arrDALI_LINE_NUM_LIGHT: ARRAY[1..2] OF BYTE := [2,1]; //korrekt rækkefølge nødvendig //rækkefølge og linje 
	arrDALI_LINE_NUM_PENDANTS: ARRAY[1..2] OF BYTE := [2,0]; //korrekt rækkefølge nødvendig. 0 = ingen pendler
END_VAR
VAR PERSISTENT
	stPirSensorData			: SH_Light.ST_DALI_Sensor;
	arrstPirSensorDataLine	: ARRAY[1..2] OF SH_Light.ST_DALI_Sensor;
	arrstTuneDataGruppe	: ARRAY [1..2] OF SH_Light.ST_TuneData_EX;
	
	uiPirOffDelayTime_MB		AT %MB34	: UINT;				//ntHMI_Pir_SetValue i gammel kode
	uiSPLuxLevel_MB			AT %MB38	: UINT;				//intHMI_Lux_SetValue i gammel kode
	uiBallastOnHours_MB		AT %MB42	: UINT;				//dintHMILysbraendtimer1 i gammel kode
	byOnHoursOverflowCount						: BYTE;
END_VAR

A_Buttons();
A_LightCtrl();
A_ModbusComm();
A_Sensor();

ACTION A_Buttons:
bTopButtonZone1		:= bTopButtonZone1_Visu;
bBottomButtonZone1	:= bBottomButtonZone1_Visu;

bButtonZone2	:= GVL_EnOcean.strEnOceanSwitch_Gang_1_216_Pendler.bT2_OFF OR GVL_EnOcean.strEnOceanSwitch_Gang_1_216_Pendler.bT2_ON;
END_ACTION

ACTION A_LightCtrl:
bNeighborRoomsPir := 	P_Gang_1_212A.stPirSensorData.bPrc OR
									P_Rum_1_213.stPirSensorData.bPrc OR
									P_Rum_1_215.stPirSensorData.bPrc OR
									P_Rum_1_217.stPirSensorData.bPrc OR
									P_Rum_1_218.stPirSensorData.bPrc OR
									P_Rum_1_219.stPirSensorData.bPrc OR
									P_Rum_1_220.stPirSensorData.bPrc OR
									P_Rum_1_222.stPirSensorData.bPrc OR
									P_Rum_1_223.stPirSensorData.bPrc OR
									GVL_AHDataModbus.arrAH_NeighborRoomsPir[5][2] OR
									GVL_AHDataModbus.arrAH_NeighborRoomsPir[5][3] OR
									GVL_AHDataModbus.arrAH_NeighborRoomsPir[5][4] OR
									GVL_AHDataModbus.arrAH_NeighborRoomsPir[5][5];

arrfbLysGruppe[1]( 
	nZoneID:= 1, 
	bButtonZone1:= bTopButtonZone1,
	bBottomButtonZone1 := bBottomButtonZone1, 
	//bTopButtonOverride := ,
	//bBottomButtonOverride := ,
	bButtonZone2:= bButtonZone2,
	//bNoButtons := ,
	bNeighborRoomsPir	:=	bNeighborRoomsPir,
	fLuxOn:= fLuxOn, 
	fLuxDim:= fLuxDim, 
	tPIRDim:= tPIRDim, 
	tPIROff:= tPIROff, 
	fOffsetSec:= fOffsetSec, 
	bReInit:= , 
	stDaliSetup:= arrstDaliSetupGruppe[1], 
	ipCommunication_Prim:= P_DALI_Background.arrfbKL6821Communication[arrDALI_LINE_NUM_LIGHT[1]], 
	//ipCommunication_Sec:= P_DALI_Background.arrfbKL6821Communication[arrDALI_LINE_NUM_LIGHT[1]],
	ipCommunication_Supl:= P_DALI_Background.arrfbKL6821Communication[arrDALI_LINE_NUM_PENDANTS[1]],
	fMinOutputPowerLevelRoom:= 15, 
	fMaxOutputPowerLevelRoom:= 100, 
	nCycleTimeInMS:= SH_Light.DALI_Param.nPlcTaskCycleTimeInMS*nDimCmdCycleTimeFactor , 
	bRunTuning:= arrRunTuningGruppe[1], 
	bOccupiedRoom=> , 
	bError_Prim=> , 
	nError_Prim=> , 
	stTuneData:=arrstTuneDataGruppe[1] , 
	stPirSensorData:= stPirSensorData, 					//samme sensordata
	stLiveData:= arrstLiveDataGruppe[1]);

	
arrfbLysGruppe[2]( 
	nZoneID:= 1, 
	bButtonZone1:= bTopButtonZone1,
	bBottomButtonZone1 := bBottomButtonZone1,
	//bTopButtonOverride := ,
	//bBottomButtonOverride := ,
	bButtonZone2:= bButtonZone2,
	//bNoButtons := ,
	bNeighborRoomsPir	:=	bNeighborRoomsPir,
	fLuxOn:= fLuxOn, 
	fLuxDim:= fLuxDim, 
	tPIRDim:= tPIRDim, 
	tPIROff:= tPIROff, 
	fOffsetSec:= fOffsetSec, 
	bReInit:= , 
	stDaliSetup:= arrstDaliSetupGruppe[2], 
	ipCommunication_Prim:= P_DALI_Background.arrfbKL6821Communication[arrDALI_LINE_NUM_LIGHT[2]], 
	//ipCommunication_Sec:= P_DALI_Background.arrfbKL6821Communication[arrDALI_LINE_NUM_LIGHT[2]],
	//ipCommunication_Supl:= P_DALI_Background.arrfbKL6821Communication[arrDALI_LINE_NUM_PENDANTS[2]],
	fMinOutputPowerLevelRoom:= 15, 
	fMaxOutputPowerLevelRoom:= 100, 
	nCycleTimeInMS:= SH_Light.DALI_Param.nPlcTaskCycleTimeInMS*nDimCmdCycleTimeFactor , 
	bRunTuning:= arrRunTuningGruppe[2], 
	bOccupiedRoom=> , 
	bError_Prim=> , 
	nError_Prim=> , 
	stTuneData:=arrstTuneDataGruppe[2] , 
	stPirSensorData:= stPirSensorData, 					//samme sensordata
	stLiveData:= arrstLiveDataGruppe[2]);
END_ACTION

ACTION A_ModbusComm:
//Manage data for modbus communication

//Manage data for read-only in PLC
stRoomDataPLC.bPirActive			:= stPirSensorData.bPrc;
stRoomDataPLC.uiActLuxLevel			:= TO_UINT(TRUNC(stPirSensorData.fBrightness));
stRoomDataPLC.uiActLightLevelPct	:= TO_UINT(TRUNC(arrfbLysGruppe[1].fbBallast.fActlLgtLvl_Prim));
		//stRoomDataPLC.uiActLightLevelPct	:= TO_UINT(TRUNC(fbLys.fbBallast.fActlLgtLvl_Prim)); //if only one group light control
stRoomDataPLC.uiBallastOnHours		:= uiBallastOnHours_MB; //The calculation for BallastOnHours is stored directly to the MB register below


//Assign data for read-only to MB registers
bPirActive_MB			:= stRoomDataPLC.bPirActive;
uiActLuxLevel_MB		:= stRoomDataPLC.uiActLuxLevel;
uiActLightLevelPct_MB	:= stRoomDataPLC.uiActLightLevelPct;

	//calculate BallastOnHours
	fbBallastOnHours(
		bEnableHourCount	:= bEnableHourCount,
		bPauseCount			:= arrfbLysGruppe[1].fbLightCtrl.bOffZone1,
		uiOnHours			:= uiBallastOnHours_MB,			//OnHours is updated here
		byOverflowCount		:= byOnHoursOverflowCount);


//Manage data for read/write for both PLC and MB registers
fbWriteSPLuxLevel(	nMaxValOut	:= uiMaxLuxLevel,
					nValIn1		:= uiSPLuxLevel_MB,		//nValIn1 takes priotity in case of download or restart
					nValIn2		:= stRoomDataPLC.uiSpLuxLevel,
					nValOut		=> uiLuxOn
				);


fbWritePirDelayTIme(	nMaxValOut	:= uiMaxPirOffMinutes,
						nValIn1		:= uiPirOffDelayTime_MB,		//nValIn1 takes priotity in case of download or restart
						nValIn2		:= stRoomDataPLC.uiPirOffDelayTime,
						nValOut		=> uiPirOffMinutes
					);
					

//Convert read/write modbus data to appropriate datatypes in PLC
fLuxOn	:= TO_REAL(uiLuxOn);			
tPIROff	:= TO_TIME(uiPirOffMinutes*udTimeScaling); //Time conversion defaults to ms

fLuxDim	:= TO_REAL(stRoomDataPLC.uiSpDimLuxLevel);			
tPIRDim	:= TO_TIME(stRoomDataPLC.uiPirDimDelayTime*udTimeScaling); //Time conversion defaults to ms
END_ACTION

ACTION A_Sensor:
fbSensor2.ipCommunication := P_DALI_Background.arrfbKL6821Communication[Sensor2_DALI_LINE_NUM];
fbSensor.ipCommunication := P_DALI_Background.arrfbKL6821Communication[Sensor_DALI_LINE_NUM];

//only 1 sensor
fbSensor2(
	byShrtAdr:= bySensor2Addr,
	bInitialize:= bInitialize2, 
	DALI_LINE_NUM:= Sensor2_DALI_LINE_NUM, 
 	//bCancelHoldTimerOccupancy:= bCancelHoldTimerOccupancy, 
	stSensorSetup := stDaliSensor2Setup,
	bInitErr=> bInitErr2, 
	bInitDone=> bInitDone2,
	stPirSensorData:= arrstPirSensorDataLine[2], 
	arrSensorScales:= arrSensor2Scales);


fbSensor(
	arrShrtAdr:= arrSensorAddr,
	bInitialize:= bInitialize, 
	DALI_LINE_NUM:= Sensor_DALI_LINE_NUM, 
 	//bCancelHoldTimerOccupancy:= bCancelHoldTimerOccupancy, 
	stSensorSetup := stDaliSensorSetup,
	arrInitErr=> arrInitErr, 
	arrInitDone=> arrInitDone,
	stPirSensorData:= arrstPirSensorDataLine[1], 
	arrSensorScales:= arrSensorScales);
	
//Input fra sensorer samles
stPirSensorData.fBrightness		:= MIN(arrstPirSensorDataLine[1].fBrightness, arrstPirSensorDataLine[2].fBrightness);
stPirSensorData.bPrc				:= arrstPirSensorDataLine[1].bPrc OR arrstPirSensorDataLine[2].bPrc;
stPirSensorData.bBrightnessRead	:= arrstPirSensorDataLine[1].bBrightnessRead OR arrstPirSensorDataLine[2].bBrightnessRead;

//Output til sensorer fordeles
IF stPirSensorData.bQueryBrightness THEN
	arrstPirSensorDataLine[1].bQueryBrightness := TRUE;
	arrstPirSensorDataLine[2].bQueryBrightness := TRUE;
ELSE
	arrstPirSensorDataLine[1].bQueryBrightness := FALSE;
	arrstPirSensorDataLine[2].bQueryBrightness := FALSE;
END_IF
END_ACTION

END_PROGRAM

// ---- POUs/Alle_Rum/Gange/Gang_1_212A/P_Gang_1_212A.TcPOU
PROGRAM P_Gang_1_212A
VAR
//Light

	fbLys			: SH_Light.FB_Light_Type_B;
	
	stDaliSetup	: SH_Light.ST_DALI_RoomSetup := (
														byShrtAdr_Prim	:= 17, 
														byGrpAdr_Prim		:= 3, 
														eMod_Prim			:= E_DALIAddressType.Group, 
														//byShrtAdr_Sec	:= 1, 
														//byGrpAdr_Sec	:= 1, 
														//eMod_Sec			:= E_DALIAddressType.Short, 
														//byShrtAdr_Supl		:= 1,
														//byGrpAdr_Supl		:= 1,
														//eMod_Supl			:= Tc3_DALI.E_DALIAddressType.Short, 
														DALI_LINE_NUM_PRIM := DALI_LINE_NUM_LIGHT, 
														DALI_LINE_NUM_SEC := 0, 
														DALI_LINE_NUM_SUPL := DALI_LINE_NUM_PENDANT);
														
	stLiveData						: SH_Light.ST_LiveData;
	bRunTuning						: BOOL;
	
	bTopButtonZone1				: BOOL;
	bTopButtonZone1_Visu		: BOOL;
	bBottomButtonZone1			: BOOL;
	bBottomButtonZone1_Visu	: BOOL;
	bButtonZone2					: BOOL;
	bNeighborRoomsPir			: BOOL;
	fLuxOn								: REAL;
	fLuxDim							: REAL;
	tPIRDim							: TIME;
	tPIROff							: TIME;
	fOffsetSec						: REAL := 20;
	bOccupiedRoom				: BOOL;
	
// Sensor Settings
	fbSensor							: SH_Light.FB_NIKO_P46xx_1Pcs;
	//fbSensor							: SH_Light.FB_NIKO_P46xx_2Pcs;
	bySensorAddr					: BYTE := 11;
	//arrSensorAddr					: ARRAY[1..2] OF BYTE := [3,4];
	bInitialize							: BOOL := TRUE;
	stDaliSensorSetup				: ST_DALI_NIKOP46SetupData := (
																nSensitivityPIRSegmentA:=bySensitivityOccupancy,
																nSensitivityPIRSegmentB:=bySensitivityOccupancy,
																nSensitivityPIRSegmentC:=bySensitivityOccupancy);
	bInitErr								: BOOL;
	bInitDone							: BOOL;
	//arrInitErr							: ARRAY [1..2] OF BOOL;
	//arrInitDone						: ARRAY [1..2] OF BOOL;
	arrSensorScales					: ARRAY [1..10] OF SH_Light.ST_DALI_SensorScaleMode :=
																						[	(fMeassureMaxSensor := rMeassure_Zone10, fReadMaxSensor := rRead_Zone10),
																							9(())];
	bCancelHoldTimerOccupancy	: BOOL;
(*	eEventPriorityOccupancy		: E_DALIEventPriority := E_DALIEVENTPRIORITY.Middle;
	nHoldTimerOccupancy			: WORD := 5; // Value in s. 	
	nReportTimerOccupancy		: BYTE := 120; // Value in s, Preset manufacturer value
	nDeadtimeTimerOccupancy		: WORD := 100; // Value in ms, Predefined Value of DALI Standard
	bCancelHoldTimerOccupancy	: BOOL;
	nSensitivityOccupancy		: BYTE:= 3; //setting Sensivity (0..4) 0 (Off), 1 (Min), 2(Low), 3(High) and 4 (Max)

	bEnableLuxEvent				: BOOL;
	eEventPriorityBrightness	: E_DALIEventPriority := E_DALIEVENTPRIORITY.Middle;
	nDeadtimeTimerBrightness	: WORD := 1500; // Value in ms, Predefined Value of DALI Standard
	nHysteresisBrightness		: BYTE := 2; // Value in %
	nHysteresisMinBrightness	: BYTE := 10; // Absolute Value, depending on the manufacturer specific resolution
	nReportTimerBrightness		: BYTE := 120; // Value in s, Preset manufacturer value
*)

//ModbusComm setup
	
	fbWriteSPLuxLevel				: SH_Light.FB_TwoVal_SelectOne_RTrigChange;
	fbWritePirDelayTIme			: SH_Light.FB_TwoVal_SelectOne_RTrigChange;
	stRoomDataPLC					: SH_Light.ST_RoomDataPLC	:=	(	uiPirOffDelayTime	:= 30,
																										uiSpLuxLevel			:= 500,
																										uiPirDimDelayTime	:= 15,
																										uiSpDimLuxLevel		:= 200);
																
	fbBallastOnHours					: SH_Light.FB_CountOnHours;
	bEnableHourCount				: BOOL := TRUE;
	
	//Non-persistent modbus data
	bPirActive_MB					AT%MX370.0	: BOOL;				//bPirLys i gammel kode
	uiActLuxLevel_MB			AT%MB374		: UINT;				//intHMIAktueltLux i gammel kode
	uiActLightLevelPct_MB	AT%MB378		: UINT;				//intDALI_Gruppe1_Lysniveau i gammel kode
	
	//For Conversion
	uiPirOffMinutes						: UINT;
	udTimeScaling						: UDINT := 60000;
	uiLuxOn								: UINT;
	
	//max values checks
	uiMaxLuxLevel						: UINT := 1023;
	uiMaxPirOffMinutes				: UINT := 180;

END_VAR

VAR CONSTANT
	Sensor_DALI_LINE_NUM			: BYTE := 2;
	DALI_LINE_NUM_LIGHT			: BYTE := 2;
	DALI_LINE_NUM_PENDANT	: BYTE := 0;
	bySensitivityOccupancy					: BYTE := 4; //setting Sensivity (0..4) 0 (Off), 1 (Min), 2(Low), 3(High) and 4 (Max)
END_VAR
VAR PERSISTENT
	stPirSensorData: SH_Light.ST_DALI_Sensor;
	stTuneData: SH_Light.ST_TuneData_EX;
	
	uiPirOffDelayTime_MB		AT%MB372	    : UINT;				//intHMI_Pir_SetValue i gammel kode
	uiSPLuxLevel_MB		    AT%MB376    	: UINT;				//intHMI_Lux_SetValue i gammel kode
	uiBallastOnHours_MB	    AT%MB380	    : UINT;				//dintHMILysbraendtimer1 i gammel kode
	byOnHoursOverflowCount			   				: BYTE;
END_VAR

A_Buttons();
A_LightCtrl();
A_ModbusComm();
A_Sensor();

ACTION A_Buttons:
bTopButtonZone1		:= 	bTopButtonZone1_Visu;
bBottomButtonZone1	:= 	bBottomButtonZone1_Visu;
END_ACTION

ACTION A_LightCtrl:
bNeighborRoomsPir := FALSE;

fbLys(
	nZoneID:= 1, 
	bButtonZone1:= bTopButtonZone1,
	bBottomButtonZone1 := bBottomButtonZone1, 
	//bButtonZone2:= bButtonZone2,
	bNeighborRoomsPir := bNeighborRoomsPir,
	fLuxOn:= fLuxOn, 
	fLuxDim:= fLuxDim, 
	tPIRDim:= tPIRDim, 
	tPIROff:= tPIROff, 
	fOffsetSec:= fOffsetSec, 
	bReInit:= , 
	stDaliSetup:= stDaliSetup, 
	ipCommunication_Prim:= P_DALI_Background.arrfbKL6821Communication[DALI_LINE_NUM_LIGHT], 
	//ipCommunication_Sec:= P_DALI_Background.arrfbKL6821Communication[DALI_LINE_NUM_LIGHT], 
	//ipCommunication_Supl:= P_DALI_Background.arrfbKL6821Communication[DALI_LINE_NUM_PENDANT],
	fMinOutputPowerLevelRoom:= 15, 
	fMaxOutputPowerLevelRoom:= 100, 
	nCycleTimeInMS:= SH_Light.DALI_Param.nPlcTaskCycleTimeInMS*nDimCmdCycleTimeFactor,  //Used only for dim. Factor=2 makes dimming smooth
	bRunTuning:= bRunTuning, 
	bOccupiedRoom=> bOccupiedRoom, 
	bError_Prim=> , 
	nError_Prim=> , 
	stTuneData:=stTuneData , 
	stPirSensorData:= stPirSensorData, 
	stLiveData:= stLiveData);
END_ACTION

ACTION A_ModbusComm:
//Manage data for modbus communication

//Manage data for read-only in PLC
stRoomDataPLC.bPirActive			:= stPirSensorData.bPrc;
stRoomDataPLC.uiActLuxLevel			:= TO_UINT(TRUNC(stPirSensorData.fBrightness));
stRoomDataPLC.uiActLightLevelPct	:= TO_UINT(TRUNC(fblys.fbBallast.fActlLgtLvl_Prim));
		//stRoomDataPLC.uiActLightLevelPct	:= TO_UINT(TRUNC(fbLys.fbBallast.fActlLgtLvl_Prim)); //if only one group light control
stRoomDataPLC.uiBallastOnHours		:= uiBallastOnHours_MB; //The calculation for BallastOnHours is stored directly to the MB register below


//Assign data for read-only to MB registers
bPirActive_MB		:= stRoomDataPLC.bPirActive;
uiActLuxLevel_MB	:= stRoomDataPLC.uiActLuxLevel;

	//calculate BallastOnHours
	fbBallastOnHours(
		bEnableHourCount	:= bEnableHourCount,
		bPauseCount			:= fbLys.fbLightCtrl.bOffZone1,
		uiOnHours			:= uiBallastOnHours_MB,			//OnHours is updated here
		byOverflowCount		:= byOnHoursOverflowCount);


//Manage data for read/write for both PLC and MB registers
fbWriteSPLuxLevel(	nMaxValOut	:= uiMaxLuxLevel,
					nValIn1		:= uiSPLuxLevel_MB,		//nValIn1 takes priotity in case of download or restart
					nValIn2		:= stRoomDataPLC.uiSpLuxLevel,
					nValOut		=> uiLuxOn
				);


fbWritePirDelayTIme(	nMaxValOut	:= uiMaxPirOffMinutes,
						nValIn1		:= uiPirOffDelayTime_MB,		//nValIn1 takes priotity in case of download or restart
						nValIn2		:= stRoomDataPLC.uiPirOffDelayTime,
						nValOut		=> uiPirOffMinutes
					);
					

//Convert read/write modbus data to appropriate datatypes in PLC
fLuxOn	:= TO_REAL(uiLuxOn);			
tPIROff	:= TO_TIME(uiPirOffMinutes*udTimeScaling); //Time conversion defaults to ms

fLuxDim	:= TO_REAL(stRoomDataPLC.uiSpDimLuxLevel);			
tPIRDim	:= TO_TIME(stRoomDataPLC.uiPirDimDelayTime*udTimeScaling); //Time conversion defaults to ms
END_ACTION

ACTION A_Sensor:

fbSensor.ipCommunication := P_DALI_Background.arrfbKL6821Communication[Sensor_DALI_LINE_NUM];


fbSensor(
	byShrtAdr:= bySensorAddr,
	bInitialize:= bInitialize, 
	DALI_LINE_NUM:= Sensor_DALI_LINE_NUM, 
 	//bCancelHoldTimerOccupancy:= bCancelHoldTimerOccupancy, 
	stSensorSetup := stDaliSensorSetup,
	bInitErr=> bInitErr, 
	bInitDone=> bInitDone,
	stPirSensorData:= stPirSensorData, 
	arrSensorScales:= arrSensorScales);


(*
fbSensor(
	arrShrtAdr:= arrSensorAddr,
	bInitialize:= bInitialize, 
	DALI_LINE_NUM:= Sensor_DALI_LINE_NUM, 
 	//bCancelHoldTimerOccupancy:= bCancelHoldTimerOccupancy, 
	stSensorSetup := stDaliSensorSetup,
	arrInitErr=> arrInitErr, 
	arrInitDone=> arrInitDone,
	stPirSensorData:= stPirSensorData, 
	arrSensorScales:= arrSensorScales);
	*)
END_ACTION

END_PROGRAM

// ---- POUs/Alle_Rum/Rum_Med_DALI_Pir/Rum_1_213/P_Rum_1_213.TcPOU
PROGRAM P_Rum_1_213
VAR
(*
Rummet består af to lysgrupper - L1G3 og L4G2 - på to forskellige linjer
Begge grupper afhænger af samme PIR-input - pir-adr. 14 og 15 - på DALI-linje 3.
Derfor oprettes to adskilte reguleringer med samme PV. Dvs., at knapfunktion og pirfunktion forbliver den samme.
*)

	arrfbLysGruppe			: ARRAY [1..2] OF FB_Light_Type_A;
	arrstDaliSetupGruppe	: ARRAY [1..2] OF SH_Light.ST_DALI_RoomSetup :=
	
													[(	byShrtAdr_Prim	:= 20, 
														byGrpAdr_Prim		:= 3, 
														eMod_Prim			:= E_DALIAddressType.Group, 
														//byShrtAdr_Sec		:= 1, 
														//byGrpAdr_Sec		:= 1, 
														//eMod_Sec			:= E_DALIAddressType.Short, 
														//byShrtAdr_Supl		:= 1,
														//byGrpAdr_Supl		:= 1,
														//eMod_Supl			:=  E_DALIAddressType.Short, 
														DALI_LINE_NUM_PRIM := arrDALI_LINE_NUM_LIGHT[1], 
														DALI_LINE_NUM_SEC := 0, //0 = ingen zonestyring/vinduerække
														DALI_LINE_NUM_SUPL := arrDALI_LINE_NUM_PENDANTS[1]),
														
													(	byShrtAdr_Prim	:= 16, 
														byGrpAdr_Prim		:= 2, 
														eMod_Prim			:= E_DALIAddressType.Group, 
														//byShrtAdr_Sec		:= 1, 
														//byGrpAdr_Sec		:= 1, 
														//eMod_Sec			:= E_DALIAddressType.Short, 
														//byShrtAdr_Supl		:= 1,
														//byGrpAdr_Supl		:= 1,
														//eMod_Supl			:=  E_DALIAddressType.Short,
														DALI_LINE_NUM_PRIM := arrDALI_LINE_NUM_LIGHT[2], 
														DALI_LINE_NUM_SEC := 0, 
														DALI_LINE_NUM_SUPL := arrDALI_LINE_NUM_PENDANTS[2])];
														
	arrstLiveDataGruppe			: ARRAY [1..2] OF SH_Light.ST_LiveData;
	arrRunTuningGruppe			: ARRAY[1..2] OF BOOL;
	
	bTopButtonZone1				: BOOL;
	bTopButtonZone1_Visu		: BOOL;
	bBottomButtonZone1			: BOOL;
	bBottomButtonZone1_Visu	: BOOL;
	bButtonZone2					: BOOL;
	bNeighborRoomsPir			: BOOL;
	fLuxOn								: REAL;
	fLuxDim							: REAL;
	tPIRDim							: TIME;
	tPIROff							: TIME;
	fOffsetSec						: REAL := 20;
	bOccupiedRoom				: BOOL;

	bRunTuning						: BOOL;


// Sensor Settings
	//fbSensor						: SH_Light.FB_NIKO_P46xx_1Pcs;
	fbSensor					: SH_Light.FB_NIKO_P46xx_2Pcs;
	//bySensorAddr				: BYTE := 7;
	arrSensorAddr			: ARRAY[1..2] OF BYTE := [14,15];
	bInitialize						: BOOL := TRUE;
	stDaliSensorSetup			: ST_DALI_NIKOP46SetupData := (
																nSensitivityPIRSegmentA:=nSensitivityOccupancy,
																nSensitivityPIRSegmentB:=nSensitivityOccupancy,
																nSensitivityPIRSegmentC:=nSensitivityOccupancy);
	//bInitErr							: BOOL;
	//bInitDone						: BOOL;
	arrInitErr						: ARRAY [1..2] OF BOOL;
	arrInitDone					: ARRAY [1..2] OF BOOL;
	arrSensorScales				: ARRAY [1..10] OF SH_Light.ST_DALI_SensorScaleMode :=
																							[	(fMeassureMaxSensor := rMeassure_Zone3, fReadMaxSensor := rRead_Zone3),
																								(fMeassureMaxSensor := rMeassure_Zone3, fReadMaxSensor := rRead_Zone3),																			
																								8(())];
																								
	bCancelHoldTimerOccupancy	: BOOL;
(*	eEventPriorityOccupancy		: E_DALIEventPriority := E_DALIEVENTPRIORITY.Middle;
	nHoldTimerOccupancy			: WORD := 5; // Value in s. 	
	nReportTimerOccupancy		: BYTE := 120; // Value in s, Preset manufacturer value
	nDeadtimeTimerOccupancy		: WORD := 100; // Value in ms, Predefined Value of DALI Standard
	bCancelHoldTimerOccupancy	: BOOL; *)
	

(*	bEnableLuxEvent				: BOOL;
	eEventPriorityBrightness	: E_DALIEventPriority := E_DALIEVENTPRIORITY.Middle;
	nDeadtimeTimerBrightness	: WORD := 1500; // Value in ms, Predefined Value of DALI Standard
	nHysteresisBrightness		: BYTE := 2; // Value in %
	nHysteresisMinBrightness	: BYTE := 10; // Absolute Value, depending on the manufacturer specific resolution
	nReportTimerBrightness		: BYTE := 120; // Value in s, Preset manufacturer value
*)

	

//ModbusComm setup
	
	fbWriteSPLuxLevel			: SH_Light.FB_TwoVal_SelectOne_RTrigChange;
	fbWritePirDelayTIme		: SH_Light.FB_TwoVal_SelectOne_RTrigChange;
	stRoomDataPLC				: SH_Light.ST_RoomDataPLC	:=	(
																	uiPirOffDelayTime	:= 30,
																	uiSpLuxLevel			:= 500,
																	uiPirDimDelayTime	:= 15,
																	uiSpDimLuxLevel		:= 200);

	fbBallastOnHours			: SH_Light.FB_CountOnHours;
	bEnableHourCount		: BOOL := TRUE;
	
	//Non-persistent modbus data
	bPirActive_MB					AT%MX0.0	: BOOL;				//bPirLys i gammel kode
	uiActLuxLevel_MB			AT%MB4		: UINT;				//intHMIAktueltLux i gammel kode
	uiActLightLevelPct_MB	AT%MB8		: UINT;				//intDALI_Gruppe1_Lysniveau i gammel kode
	
	//For Conversion
	uiPirOffMinutes						: UINT;
	udTimeScaling						: UDINT := 60000;
	uiLuxOn								: UINT;
	
	//max values checks
	uiMaxLuxLevel						: UINT := 1023;
	uiMaxPirOffMinutes				: UINT := 180;


END_VAR

VAR CONSTANT
	Sensor_DALI_LINE_NUM				: BYTE := 3;
	arrDALI_LINE_NUM_LIGHT			: ARRAY[1..2] OF BYTE := [1,4]; //korrekt rækkefølge nødvendig
	arrDALI_LINE_NUM_PENDANTS: ARRAY[1..2] OF BYTE := [0,0]; //korrekt rækkefølge nødvendig. 0 = ingen pendler
	nSensitivityOccupancy						: BYTE:= 3; //setting Sensivity (0..4) 0 (Off), 1 (Min), 2(Low), 3(High) and 4 (Max)
END_VAR

VAR PERSISTENT
	stPirSensorData: SH_Light.ST_DALI_Sensor;
	arrstTuneDataGruppe: ARRAY [1..2] OF SH_Light.ST_TuneData_EX;
	
	uiPirOffDelayTime_MB		AT%MB2			: UINT;				//intHMI_Pir_SetValue i gammel kode
	uiSPLuxLevel_MB			AT%MB6			: UINT;				//intHMI_Lux_SetValue i gammel kode
	uiBallastOnHours_MB		AT%MB10		: UINT;				//dintHMILysbraendtimer1 i gammel kode
   	byOnHoursOverflowCount							: BYTE;
END_VAR

A_Buttons();
A_LightCtrl();
A_Sensor();
A_modbuscomm();

ACTION A_Buttons:
bTopButtonZone1		:= GVL_EnOcean.strEnOceanSwitch_Rum_1_213_Indgang.bT2_ON OR GVL_EnOcean.strEnOceanSwitch_Rum_1_213_Ekstra.bT1_ON OR bTopButtonZone1_Visu;
bBottomButtonZone1	:= GVL_EnOcean.strEnOceanSwitch_Rum_1_213_Indgang.bT2_OFF OR  GVL_EnOcean.strEnOceanSwitch_Rum_1_213_Ekstra.bT1_OFF OR bBottomButtonZone1_Visu;
END_ACTION

ACTION A_LightCtrl:

arrfbLysGruppe[1]( 
	nZoneID:= 1, 
	bButtonZone1:= bTopButtonZone1,
	bBottomButtonZone1 := bBottomButtonZone1, 
	//bButtonZone2:= bButtonZone2,
	fLuxOn:= fLuxOn, 
	fLuxDim:= fLuxDim, 
	tPIRDim:= tPIRDim, 
	tPIROff:= tPIROff, 
	fOffsetSec:= fOffsetSec, 
	bReInit:= , 
	stDaliSetup:= arrstDaliSetupGruppe[1], 
	ipCommunication_Prim:= P_DALI_Background.arrfbKL6821Communication[arrDALI_LINE_NUM_LIGHT[1]], 
	//ipCommunication_Sec:= P_DALI_Background.arrfbKL6821Communication[arrDALI_LINE_NUM_LIGHT[1]],
	//ipCommunication_Supl:= P_DALI_Background.arrfbKL6821Communication[arrDALI_LINE_NUM_PENDANTS[1]],
	fMinOutputPowerLevelRoom:= 15, 
	fMaxOutputPowerLevelRoom:= 100, 
	nCycleTimeInMS:= SH_Light.DALI_Param.nPlcTaskCycleTimeInMS*SH_Light.DALI_Param.nDimCmdCycleTimeFactor, 
	bRunTuning:= arrRunTuningGruppe[1], 
	bOccupiedRoom=> , 
	bError_Prim=> , 
	nError_Prim=> , 
	stTuneData:=arrstTuneDataGruppe[1] , 
	stPirSensorData:= stPirSensorData, 					//samme sensordata
	stLiveData:= arrstLiveDataGruppe[1]);

arrfbLysGruppe[2]( 
	nZoneID:= 1, 
	bButtonZone1:= bTopButtonZone1,
	bBottomButtonZone1 := bBottomButtonZone1, 
	bButtonZone2:= bButtonZone2,
	fLuxOn:= fLuxOn, 
	fLuxDim:= fLuxDim, 
	tPIRDim:= tPIRDim, 
	tPIROff:= tPIROff, 
	fOffsetSec:= fOffsetSec, 
	bReInit:= , 
	stDaliSetup:= arrstDaliSetupGruppe[2], 
	ipCommunication_Prim:= P_DALI_Background.arrfbKL6821Communication[arrDALI_LINE_NUM_LIGHT[2]], 
	//ipCommunication_Sec:= P_DALI_Background.arrfbKL6821Communication[arrDALI_LINE_NUM_LIGHT[2]],
	//ipCommunication_Supl:= P_DALI_Background.arrfbKL6821Communication[arrDALI_LINE_NUM_PENDANTS[2]],
	fMinOutputPowerLevelRoom:= 15, 
	fMaxOutputPowerLevelRoom:= 100, 
	nCycleTimeInMS:= SH_Light.DALI_Param.nPlcTaskCycleTimeInMS*SH_Light.DALI_Param.nDimCmdCycleTimeFactor, 
	bRunTuning:= arrRunTuningGruppe[2], 
	bOccupiedRoom=> , 
	bError_Prim=> , 
	nError_Prim=> , 
	stTuneData:=arrstTuneDataGruppe[2] , 
	stPirSensorData:= stPirSensorData, 					//samme sensordata
	stLiveData:= arrstLiveDataGruppe[2]);
END_ACTION

ACTION A_ModbusComm:
//Manage data for modbus communication

//Manage data for read-only in PLC
stRoomDataPLC.bPirActive			:= stPirSensorData.bPrc;
stRoomDataPLC.uiActLuxLevel			:= TO_UINT(TRUNC(stPirSensorData.fBrightness));
stRoomDataPLC.uiActLightLevelPct	:= TO_UINT(TRUNC(arrfbLysGruppe[1].fbBallast.fActlLgtLvl_Prim));
		//stRoomDataPLC.uiActLightLevelPct	:= TO_UINT(TRUNC(fbLys.fbBallast.fActlLgtLvl_Prim)); //if only one group light control
stRoomDataPLC.uiBallastOnHours		:= uiBallastOnHours_MB; //The calculation for BallastOnHours is stored directly to the MB register below


//Assign data for read-only to MB registers
bPirActive_MB			:= stRoomDataPLC.bPirActive;
uiActLuxLevel_MB		:= stRoomDataPLC.uiActLuxLevel;
uiActLightLevelPct_MB	:= stRoomDataPLC.uiActLightLevelPct;

	//calculate BallastOnHours
	fbBallastOnHours(
		bEnableHourCount	:= bEnableHourCount,
		bPauseCount			:= arrfbLysGruppe[1].fbLightCtrl.bOffZone1,
		uiOnHours			:= uiBallastOnHours_MB,			//OnHours is updated here
		byOverflowCount		:= byOnHoursOverflowCount);


//Manage data for read/write for both PLC and MB registers
fbWriteSPLuxLevel(	nMaxValOut	:= uiMaxLuxLevel,
					nValIn1		:= uiSPLuxLevel_MB,		//nValIn1 takes priotity in case of download or restart
					nValIn2		:= stRoomDataPLC.uiSpLuxLevel,
					nValOut		=> uiLuxOn
				);


fbWritePirDelayTIme(	nMaxValOut	:= uiMaxPirOffMinutes,
						nValIn1		:= uiPirOffDelayTime_MB,		//nValIn1 takes priotity in case of download or restart
						nValIn2		:= stRoomDataPLC.uiPirOffDelayTime,
						nValOut		=> uiPirOffMinutes
					);
					

//Convert read/write modbus data to appropriate datatypes in PLC
fLuxOn	:= TO_REAL(uiLuxOn);			
tPIROff	:= TO_TIME(uiPirOffMinutes*udTimeScaling); //Time conversion defaults to ms

fLuxDim	:= TO_REAL(stRoomDataPLC.uiSpDimLuxLevel);			
tPIRDim	:= TO_TIME(stRoomDataPLC.uiPirDimDelayTime*udTimeScaling); //Time conversion defaults to ms
END_ACTION

ACTION A_Sensor:

fbSensor.ipCommunication := P_DALI_Background.arrfbKL6821Communication[Sensor_DALI_LINE_NUM];
(*
//only 1 sensor
fbSensor(
	byShrtAdr:= bySensorAddr,
	bInitialize:= bInitialize, 
	DALI_LINE_NUM:= Sensor_DALI_LINE_NUM, 
 	//bCancelHoldTimerOccupancy:= bCancelHoldTimerOccupancy, 
	stSensorSetup := stDaliSensorSetup,
	bInitErr=> bInitErr, 
	bInitDone=> bInitDone,
	stPirSensorData:= stPirSensorData, 
	arrSensorScales:= arrSensorScales);
	*)
	

//several sensors	
fbSensor(
	arrShrtAdr:= arrSensorAddr,
	bInitialize:= bInitialize, 
	DALI_LINE_NUM:= Sensor_DALI_LINE_NUM, 
 	//bCancelHoldTimerOccupancy:= bCancelHoldTimerOccupancy, 
	stSensorSetup := stDaliSensorSetup,
	arrInitErr=> arrInitErr, 
	arrInitDone=> arrInitDone,
	stPirSensorData:= stPirSensorData, 
	arrSensorScales:= arrSensorScales);
END_ACTION

END_PROGRAM

// ---- POUs/Alle_Rum/Rum_Med_DALI_Pir/Rum_1_215/P_Rum_1_215.TcPOU
PROGRAM P_Rum_1_215
VAR
//Light

	fbLys			: FB_Light_Type_A;
	
	stDaliSetup	: SH_Light.ST_DALI_RoomSetup := (
														byShrtAdr_Prim	:= 20, 
														byGrpAdr_Prim		:= 3, 
														eMod_Prim			:= E_DALIAddressType.Group, 
														//byShrtAdr_Sec	:= 1, 
														//byGrpAdr_Sec	:= 1, 
														//eMod_Sec			:= E_DALIAddressType.Short, 
														//byShrtAdr_Supl		:= 1,
														//byGrpAdr_Supl		:= 1,
														//eMod_Supl			:= Tc3_DALI.E_DALIAddressType.Short, 
														DALI_LINE_NUM_PRIM := DALI_LINE_NUM_LIGHT, 
														DALI_LINE_NUM_SEC := 0, 
														DALI_LINE_NUM_SUPL := DALI_LINE_NUM_PENDANT);
														
	stLiveData					: SH_Light.ST_LiveData;
	bRunTuning					: BOOL;
	
	bTopButtonZone1			: BOOL;
	bTopButtonZone1_Visu	: BOOL;
	bBottomButtonZone1		: BOOL;
	bBottomButtonZone1_Visu	: BOOL;
	bButtonZone2				: BOOL;
	fLuxOn							: REAL;
	fLuxDim						: REAL;
	tPIRDim						: TIME;
	tPIROff						: TIME;
	fOffsetSec					: REAL := 20;
	bOccupiedRoom			: BOOL;
	
// Sensor Settings
	fbSensor						: SH_Light.FB_NIKO_P46xx_1Pcs;
	//fbSensor						: SH_Light.FB_NIKO_P46xx_2Pcs;
	bySensorAddr				: BYTE := 5;
	//arrSensorAddr				: ARRAY[1..2] OF BYTE := [4,5];
	bInitialize						: BOOL := TRUE;
	stDaliSensorSetup			: ST_DALI_NIKOP46SetupData;
	bInitErr							: BOOL;
	bInitDone						: BOOL;
	//arrInitErr						: ARRAY [1..2] OF BOOL;
	//arrInitDone					: ARRAY [1..2] OF BOOL;
	arrSensorScales				: ARRAY [1..10] OF SH_Light.ST_DALI_SensorScaleMode :=
																						[	(fMeassureMaxSensor := rMeassure_Zone3, fReadMaxSensor := rRead_Zone3),	
																							9(())];
	bCancelHoldTimerOccupancy	: BOOL;
(*	eEventPriorityOccupancy		: E_DALIEventPriority := E_DALIEVENTPRIORITY.Middle;
	nHoldTimerOccupancy			: WORD := 5; // Value in s. 	
	nReportTimerOccupancy		: BYTE := 120; // Value in s, Preset manufacturer value
	nDeadtimeTimerOccupancy		: WORD := 100; // Value in ms, Predefined Value of DALI Standard
	bCancelHoldTimerOccupancy	: BOOL;
	nSensitivityOccupancy		: BYTE:= 3; //setting Sensivity (0..4) 0 (Off), 1 (Min), 2(Low), 3(High) and 4 (Max)

	bEnableLuxEvent				: BOOL;
	eEventPriorityBrightness	: E_DALIEventPriority := E_DALIEVENTPRIORITY.Middle;
	nDeadtimeTimerBrightness	: WORD := 1500; // Value in ms, Predefined Value of DALI Standard
	nHysteresisBrightness		: BYTE := 2; // Value in %
	nHysteresisMinBrightness	: BYTE := 10; // Absolute Value, depending on the manufacturer specific resolution
	nReportTimerBrightness		: BYTE := 120; // Value in s, Preset manufacturer value
*)

//ModbusComm setup
	
	fbWriteSPLuxLevel				: SH_Light.FB_TwoVal_SelectOne_RTrigChange;
	fbWritePirDelayTIme			: SH_Light.FB_TwoVal_SelectOne_RTrigChange;
	stRoomDataPLC					: SH_Light.ST_RoomDataPLC	:=	(	uiPirOffDelayTime	:= 30,
																										uiSpLuxLevel			:= 500,
																										uiPirDimDelayTime	:= 15,
																										uiSpDimLuxLevel		:= 200);
																
	fbBallastOnHours					: SH_Light.FB_CountOnHours;
	bEnableHourCount				: BOOL := TRUE;
	
	//Non-persistent modbus data
	bPirActive_MB					AT%MX16.0	: BOOL;				//bPirLys i gammel kode
	uiActLuxLevel_MB			AT%MB20		: UINT;				//intHMIAktueltLux i gammel kode
	uiActLightLevelPct_MB	AT%MB24		: UINT;				//intDALI_Gruppe1_Lysniveau i gammel kode
	
	//For Conversion
	uiPirOffMinutes						: UINT;
	udTimeScaling						: UDINT := 60000;
	uiLuxOn								: UINT;
	
	//max values checks
	uiMaxLuxLevel						: UINT := 1023;
	uiMaxPirOffMinutes				: UINT := 180;

END_VAR

VAR CONSTANT
	Sensor_DALI_LINE_NUM: BYTE := 4;
	DALI_LINE_NUM_LIGHT: BYTE := 4;
	DALI_LINE_NUM_PENDANT: BYTE :=0;
END_VAR
VAR PERSISTENT
	stPirSensorData: SH_Light.ST_DALI_Sensor;
	stTuneData: SH_Light.ST_TuneData_EX;
	
	uiPirOffDelayTime_MB		AT%MB18	    	: UINT;				//intHMI_Pir_SetValue i gammel kode
	uiSPLuxLevel_MB		    AT%MB22    		: UINT;				//intHMI_Lux_SetValue i gammel kode
	uiBallastOnHours_MB	    AT%MB26		    : UINT;				//dintHMILysbraendtimer1 i gammel kode
	byOnHoursOverflowCount			   					: BYTE;
END_VAR

A_Buttons();
A_LightCtrl();
A_ModbusComm();
A_Sensor();

ACTION A_Buttons:
bTopButtonZone1		:= GVL_EnOcean.strEnOceanSwitch_Rum_1_215.bT2_OFF OR
									bTopButtonZone1_Visu;
bBottomButtonZone1	:= GVL_EnOcean.strEnOceanSwitch_Rum_1_215.bT2_ON OR
									bBottomButtonZone1_Visu;
END_ACTION

ACTION A_LightCtrl:

fbLys(
	nZoneID:= 1, 
	bButtonZone1:= bTopButtonZone1,
	bBottomButtonZone1 := bBottomButtonZone1, 
	//bButtonZone2:= bButtonZone2, 
	fLuxOn:= fLuxOn, 
	fLuxDim:= fLuxDim, 
	tPIRDim:= tPIRDim, 
	tPIROff:= tPIROff, 
	fOffsetSec:= fOffsetSec, 
	bReInit:= , 
	stDaliSetup:= stDaliSetup, 
	ipCommunication_Prim:= P_DALI_Background.arrfbKL6821Communication[DALI_LINE_NUM_LIGHT], 
	//ipCommunication_Sec:= P_DALI_Background.arrfbKL6821Communication[DALI_LINE_NUM_LIGHT], 
	//ipCommunication_Supl:= P_DALI_Background.arrfbKL6821Communication[DALI_LINE_NUM_PENDANT],
	fMinOutputPowerLevelRoom:= 15, 
	fMaxOutputPowerLevelRoom:= 100, 
	nCycleTimeInMS:= SH_Light.DALI_Param.nPlcTaskCycleTimeInMS*nDimCmdCycleTimeFactor,
	bRunTuning:= bRunTuning, 
	bOccupiedRoom=> bOccupiedRoom, 
	bError_Prim=> , 
	nError_Prim=> , 
	stTuneData:=stTuneData , 
	stPirSensorData:= stPirSensorData, 
	stLiveData:= stLiveData);
END_ACTION

ACTION A_ModbusComm:
//Manage data for modbus communication

//Manage data for read-only in PLC
stRoomDataPLC.bPirActive			:= stPirSensorData.bPrc;
stRoomDataPLC.uiActLuxLevel			:= TO_UINT(TRUNC(stPirSensorData.fBrightness));
stRoomDataPLC.uiActLightLevelPct	:= TO_UINT(TRUNC(fblys.fbBallast.fActlLgtLvl_Prim));
		//stRoomDataPLC.uiActLightLevelPct	:= TO_UINT(TRUNC(fbLys.fbBallast.fActlLgtLvl_Prim)); //if only one group light control
stRoomDataPLC.uiBallastOnHours		:= uiBallastOnHours_MB; //The calculation for BallastOnHours is stored directly to the MB register below


//Assign data for read-only to MB registers
bPirActive_MB		:= stRoomDataPLC.bPirActive;
uiActLuxLevel_MB	:= stRoomDataPLC.uiActLuxLevel;

	//calculate BallastOnHours
	fbBallastOnHours(
		bEnableHourCount	:= bEnableHourCount,
		bPauseCount			:= fbLys.fbLightCtrl.bOffZone1,
		uiOnHours			:= uiBallastOnHours_MB,			//OnHours is updated here
		byOverflowCount		:= byOnHoursOverflowCount);


//Manage data for read/write for both PLC and MB registers
fbWriteSPLuxLevel(	nMaxValOut	:= uiMaxLuxLevel,
					nValIn1		:= uiSPLuxLevel_MB,		//nValIn1 takes priotity in case of download or restart
					nValIn2		:= stRoomDataPLC.uiSpLuxLevel,
					nValOut		=> uiLuxOn
				);


fbWritePirDelayTIme(	nMaxValOut	:= uiMaxPirOffMinutes,
						nValIn1		:= uiPirOffDelayTime_MB,		//nValIn1 takes priotity in case of download or restart
						nValIn2		:= stRoomDataPLC.uiPirOffDelayTime,
						nValOut		=> uiPirOffMinutes
					);
					

//Convert read/write modbus data to appropriate datatypes in PLC
fLuxOn	:= TO_REAL(uiLuxOn);			
tPIROff	:= TO_TIME(uiPirOffMinutes*udTimeScaling); //Time conversion defaults to ms

fLuxDim	:= TO_REAL(stRoomDataPLC.uiSpDimLuxLevel);			
tPIRDim	:= TO_TIME(stRoomDataPLC.uiPirDimDelayTime*udTimeScaling); //Time conversion defaults to ms
END_ACTION

ACTION A_Sensor:

fbSensor.ipCommunication := P_DALI_Background.arrfbKL6821Communication[Sensor_DALI_LINE_NUM];

//Only one sensor
fbSensor(
	byShrtAdr:= bySensorAddr,
	bInitialize:= bInitialize, 
	DALI_LINE_NUM:= Sensor_DALI_LINE_NUM, 
 	//bCancelHoldTimerOccupancy:= bCancelHoldTimerOccupancy, 
	stSensorSetup := stDaliSensorSetup,
	bInitErr=> bInitErr, 
	bInitDone=> bInitDone,
	stPirSensorData:= stPirSensorData, 
	arrSensorScales:= arrSensorScales);
	

(*
//Several sensors
fbSensor(
	arrShrtAdr:= arrSensorAddr,
	bInitialize:= bInitialize, 
	DALI_LINE_NUM:= Sensor_DALI_LINE_NUM, 
 	//bCancelHoldTimerOccupancy:= bCancelHoldTimerOccupancy, 
	stSensorSetup := stDaliSensorSetup,
	arrInitErr=> arrInitErr, 
	arrInitDone=> arrInitDone,
	stPirSensorData:= stPirSensorData, 
	arrSensorScales:= arrSensorScales);
	*)
END_ACTION

END_PROGRAM

// ---- POUs/Alle_Rum/Rum_Med_DALI_Pir/Rum_1_217/P_Rum_1_217.TcPOU
PROGRAM P_Rum_1_217
VAR
(*
Rummet består af en lysgruppe og et ekstra armatur - L1G4 og L4S22 - på to forskellige linjer
Både gruppen og ekstra armatur afhænger af samme PIR-input - pir-adr. 3 - på DALI-linje 4.
Derfor oprettes to adskilte reguleringer med samme PV. Dvs., at knapfunktion og pirfunktion forbliver den samme.
*)

	arrfbLysGruppe			: ARRAY [1..2] OF FB_Light_Type_A;
	arrstDaliSetupGruppe	: ARRAY [1..2] OF SH_Light.ST_DALI_RoomSetup :=
	
													[(	byShrtAdr_Prim	:= 22, 
														byGrpAdr_Prim		:= 4, 
														eMod_Prim			:= E_DALIAddressType.Group, 
														//byShrtAdr_Sec		:= 1, 
														//byGrpAdr_Sec		:= 1, 
														//eMod_Sec			:= E_DALIAddressType.Short, 
														//byShrtAdr_Supl		:= 1,
														//byGrpAdr_Supl		:= 1,
														//eMod_Supl			:=  E_DALIAddressType.Short, 
														DALI_LINE_NUM_PRIM := arrDALI_LINE_NUM_LIGHT[1], 
														DALI_LINE_NUM_SEC := 0, //0 = ingen zonestyring/vinduerække
														DALI_LINE_NUM_SUPL := arrDALI_LINE_NUM_PENDANTS[1]),
														
													(	byShrtAdr_Prim	:= 22, 
														//byGrpAdr_Prim		:= 1, 
														eMod_Prim			:= E_DALIAddressType.Short, 
														//byShrtAdr_Sec		:= 1, 
														//byGrpAdr_Sec		:= 1, 
														//eMod_Sec			:= E_DALIAddressType.Short, 
														//byShrtAdr_Supl		:= 1,
														//byGrpAdr_Supl		:= 1,
														//eMod_Supl			:=  E_DALIAddressType.Short,
														DALI_LINE_NUM_PRIM := arrDALI_LINE_NUM_LIGHT[2], 
														DALI_LINE_NUM_SEC := 0, 
														DALI_LINE_NUM_SUPL := arrDALI_LINE_NUM_PENDANTS[2])];
														
	arrstLiveDataGruppe			: ARRAY [1..2] OF SH_Light.ST_LiveData;
	arrRunTuningGruppe			: ARRAY[1..2] OF BOOL;
	
	bTopButtonZone1				: BOOL;
	bTopButtonZone1_Visu		: BOOL;
	bBottomButtonZone1			: BOOL;
	bBottomButtonZone1_Visu	: BOOL;
	bButtonZone2					: BOOL;
	bNeighborRoomsPir			: BOOL;
	fLuxOn								: REAL;
	fLuxDim							: REAL;
	tPIRDim							: TIME;
	tPIROff							: TIME;
	fOffsetSec						: REAL := 20;
	bOccupiedRoom				: BOOL;

	bRunTuning						: BOOL;


// Sensor Settings
	fbSensor						: SH_Light.FB_NIKO_P46xx_1Pcs;
	//fbSensor					: SH_Light.FB_NIKO_P46xx_3Pcs;
	bySensorAddr				: BYTE := 3;
	//arrSensorAddr			: ARRAY[1..3] OF BYTE := [7,8,9];
	bInitialize						: BOOL := TRUE;
	stDaliSensorSetup			: ST_DALI_NIKOP46SetupData := (
																nSensitivityPIRSegmentA:=nSensitivityOccupancy,
																nSensitivityPIRSegmentB:=nSensitivityOccupancy,
																nSensitivityPIRSegmentC:=nSensitivityOccupancy);
	bInitErr							: BOOL;
	bInitDone						: BOOL;
	//arrInitErr					: ARRAY [1..3] OF BOOL;
	//arrInitDone				: ARRAY [1..3] OF BOOL;
	arrSensorScales				: ARRAY [1..10] OF SH_Light.ST_DALI_SensorScaleMode :=
																							[	(fMeassureMaxSensor := rMeassure_Zone3, fReadMaxSensor := rRead_Zone3),																							
																								9(())];
																								
	bCancelHoldTimerOccupancy	: BOOL;
(*	eEventPriorityOccupancy		: E_DALIEventPriority := E_DALIEVENTPRIORITY.Middle;
	nHoldTimerOccupancy			: WORD := 5; // Value in s. 	
	nReportTimerOccupancy		: BYTE := 120; // Value in s, Preset manufacturer value
	nDeadtimeTimerOccupancy		: WORD := 100; // Value in ms, Predefined Value of DALI Standard
	bCancelHoldTimerOccupancy	: BOOL; *)
	

(*	bEnableLuxEvent				: BOOL;
	eEventPriorityBrightness	: E_DALIEventPriority := E_DALIEVENTPRIORITY.Middle;
	nDeadtimeTimerBrightness	: WORD := 1500; // Value in ms, Predefined Value of DALI Standard
	nHysteresisBrightness		: BYTE := 2; // Value in %
	nHysteresisMinBrightness	: BYTE := 10; // Absolute Value, depending on the manufacturer specific resolution
	nReportTimerBrightness		: BYTE := 120; // Value in s, Preset manufacturer value
*)

	

//ModbusComm setup
	
	fbWriteSPLuxLevel			: SH_Light.FB_TwoVal_SelectOne_RTrigChange;
	fbWritePirDelayTIme		: SH_Light.FB_TwoVal_SelectOne_RTrigChange;
	stRoomDataPLC				: SH_Light.ST_RoomDataPLC	:=	(
																	uiPirOffDelayTime	:= 30,
																	uiSpLuxLevel			:= 500,
																	uiPirDimDelayTime	:= 15,
																	uiSpDimLuxLevel		:= 200);

	fbBallastOnHours			: SH_Light.FB_CountOnHours;
	bEnableHourCount		: BOOL := TRUE;
	
	//Non-persistent modbus data
	bPirActive_MB					AT%MX48.0	: BOOL;				//bPirLys i gammel kode
	uiActLuxLevel_MB			AT%MB52		: UINT;				//intHMIAktueltLux i gammel kode
	uiActLightLevelPct_MB	AT%MB56		: UINT;				//intDALI_Gruppe1_Lysniveau i gammel kode
	
	//For Conversion
	uiPirOffMinutes						: UINT;
	udTimeScaling						: UDINT := 60000;
	uiLuxOn								: UINT;
	
	//max values checks
	uiMaxLuxLevel						: UINT := 1023;
	uiMaxPirOffMinutes				: UINT := 180;


END_VAR

VAR CONSTANT
	Sensor_DALI_LINE_NUM				: BYTE := 4;
	arrDALI_LINE_NUM_LIGHT			: ARRAY[1..2] OF BYTE := [1,4]; //korrekt rækkefølge nødvendig
	arrDALI_LINE_NUM_PENDANTS: ARRAY[1..2] OF BYTE := [0,0]; //korrekt rækkefølge nødvendig. 0 = ingen pendler
	nSensitivityOccupancy						: BYTE:= 4; //setting Sensivity (0..4) 0 (Off), 1 (Min), 2(Low), 3(High) and 4 (Max)
END_VAR

VAR PERSISTENT
	stPirSensorData: SH_Light.ST_DALI_Sensor;
	arrstTuneDataGruppe: ARRAY [1..2] OF SH_Light.ST_TuneData_EX;
	
	uiPirOffDelayTime_MB		AT%MB50	    : UINT;				//intHMI_Pir_SetValue i gammel kode
	uiSPLuxLevel_MB			AT%MB54	    : UINT;				//intHMI_Lux_SetValue i gammel kode
	uiBallastOnHours_MB		AT%MB58		: UINT;				//dintHMILysbraendtimer1 i gammel kode
   	byOnHoursOverflowCount							: BYTE;
END_VAR

A_Buttons();
A_LightCtrl();
A_Sensor();
A_modbuscomm();

ACTION A_Buttons:
bTopButtonZone1		:= GVL_EnOcean.strEnOceanSwitch_Rum_1_217.bT1_ON OR bTopButtonZone1_Visu;
bBottomButtonZone1	:= GVL_EnOcean.strEnOceanSwitch_Rum_1_217.bT1_OFF OR bBottomButtonZone1_Visu;
END_ACTION

ACTION A_LightCtrl:
//Linje 2
arrfbLysGruppe[1]( 
	nZoneID:= 1, 
	bButtonZone1:= bTopButtonZone1,
	bBottomButtonZone1 := bBottomButtonZone1, 
	//bButtonZone2:= bButtonZone2,
	fLuxOn:= fLuxOn, 
	fLuxDim:= fLuxDim, 
	tPIRDim:= tPIRDim, 
	tPIROff:= tPIROff, 
	fOffsetSec:= fOffsetSec, 
	bReInit:= , 
	stDaliSetup:= arrstDaliSetupGruppe[1], 
	ipCommunication_Prim:= P_DALI_Background.arrfbKL6821Communication[arrDALI_LINE_NUM_LIGHT[1]], 
	//ipCommunication_Sec:= P_DALI_Background.arrfbKL6821Communication[arrDALI_LINE_NUM_LIGHT[1]],
	//ipCommunication_Supl:= P_DALI_Background.arrfbKL6821Communication[arrDALI_LINE_NUM_PENDANTS[1]],
	fMinOutputPowerLevelRoom:= 15, 
	fMaxOutputPowerLevelRoom:= 100, 
	nCycleTimeInMS:= SH_Light.DALI_Param.nPlcTaskCycleTimeInMS*SH_Light.DALI_Param.nDimCmdCycleTimeFactor, 
	bRunTuning:= arrRunTuningGruppe[1], 
	bOccupiedRoom=> , 
	bError_Prim=> , 
	nError_Prim=> , 
	stTuneData:=arrstTuneDataGruppe[1] , 
	stPirSensorData:= stPirSensorData, 					//samme sensordata
	stLiveData:= arrstLiveDataGruppe[1]);

//Linje 1 
arrfbLysGruppe[2]( 
	nZoneID:= 1, 
	bButtonZone1:= bTopButtonZone1,
	bBottomButtonZone1 := bBottomButtonZone1, 
	bButtonZone2:= bButtonZone2,
	fLuxOn:= fLuxOn, 
	fLuxDim:= fLuxDim, 
	tPIRDim:= tPIRDim, 
	tPIROff:= tPIROff, 
	fOffsetSec:= fOffsetSec, 
	bReInit:= , 
	stDaliSetup:= arrstDaliSetupGruppe[2], 
	ipCommunication_Prim:= P_DALI_Background.arrfbKL6821Communication[arrDALI_LINE_NUM_LIGHT[2]], 
	//ipCommunication_Sec:= P_DALI_Background.arrfbKL6821Communication[arrDALI_LINE_NUM_LIGHT[2]],
	//ipCommunication_Supl:= P_DALI_Background.arrfbKL6821Communication[arrDALI_LINE_NUM_PENDANTS[2]],
	fMinOutputPowerLevelRoom:= 15, 
	fMaxOutputPowerLevelRoom:= 100, 
	nCycleTimeInMS:= SH_Light.DALI_Param.nPlcTaskCycleTimeInMS*SH_Light.DALI_Param.nDimCmdCycleTimeFactor, 
	bRunTuning:= arrRunTuningGruppe[2], 
	bOccupiedRoom=> , 
	bError_Prim=> , 
	nError_Prim=> , 
	stTuneData:=arrstTuneDataGruppe[2] , 
	stPirSensorData:= stPirSensorData, 					//samme sensordata
	stLiveData:= arrstLiveDataGruppe[2]);
END_ACTION

ACTION A_ModbusComm:
//Manage data for modbus communication

//Manage data for read-only in PLC
stRoomDataPLC.bPirActive			:= stPirSensorData.bPrc;
stRoomDataPLC.uiActLuxLevel			:= TO_UINT(TRUNC(stPirSensorData.fBrightness));
stRoomDataPLC.uiActLightLevelPct	:= TO_UINT(TRUNC(arrfbLysGruppe[1].fbBallast.fActlLgtLvl_Prim));
		//stRoomDataPLC.uiActLightLevelPct	:= TO_UINT(TRUNC(fbLys.fbBallast.fActlLgtLvl_Prim)); //if only one group light control
stRoomDataPLC.uiBallastOnHours		:= uiBallastOnHours_MB; //The calculation for BallastOnHours is stored directly to the MB register below


//Assign data for read-only to MB registers
bPirActive_MB			:= stRoomDataPLC.bPirActive;
uiActLuxLevel_MB		:= stRoomDataPLC.uiActLuxLevel;
uiActLightLevelPct_MB	:= stRoomDataPLC.uiActLightLevelPct;

	//calculate BallastOnHours
	fbBallastOnHours(
		bEnableHourCount	:= bEnableHourCount,
		bPauseCount			:= arrfbLysGruppe[1].fbLightCtrl.bOffZone1,
		uiOnHours			:= uiBallastOnHours_MB,			//OnHours is updated here
		byOverflowCount		:= byOnHoursOverflowCount);


//Manage data for read/write for both PLC and MB registers
fbWriteSPLuxLevel(	nMaxValOut	:= uiMaxLuxLevel,
					nValIn1		:= uiSPLuxLevel_MB,		//nValIn1 takes priotity in case of download or restart
					nValIn2		:= stRoomDataPLC.uiSpLuxLevel,
					nValOut		=> uiLuxOn
				);


fbWritePirDelayTIme(	nMaxValOut	:= uiMaxPirOffMinutes,
						nValIn1		:= uiPirOffDelayTime_MB,		//nValIn1 takes priotity in case of download or restart
						nValIn2		:= stRoomDataPLC.uiPirOffDelayTime,
						nValOut		=> uiPirOffMinutes
					);
					

//Convert read/write modbus data to appropriate datatypes in PLC
fLuxOn	:= TO_REAL(uiLuxOn);			
tPIROff	:= TO_TIME(uiPirOffMinutes*udTimeScaling); //Time conversion defaults to ms

fLuxDim	:= TO_REAL(stRoomDataPLC.uiSpDimLuxLevel);			
tPIRDim	:= TO_TIME(stRoomDataPLC.uiPirDimDelayTime*udTimeScaling); //Time conversion defaults to ms
END_ACTION

ACTION A_Sensor:

fbSensor.ipCommunication := P_DALI_Background.arrfbKL6821Communication[Sensor_DALI_LINE_NUM];

//only 1 sensor
fbSensor(
	byShrtAdr:= bySensorAddr,
	bInitialize:= bInitialize, 
	DALI_LINE_NUM:= Sensor_DALI_LINE_NUM, 
 	//bCancelHoldTimerOccupancy:= bCancelHoldTimerOccupancy, 
	stSensorSetup := stDaliSensorSetup,
	bInitErr=> bInitErr, 
	bInitDone=> bInitDone,
	stPirSensorData:= stPirSensorData, 
	arrSensorScales:= arrSensorScales);
	
(*//
//several sensors	
fbSensor(
	arrShrtAdr:= arrSensorAddr,
	bInitialize:= bInitialize, 
	DALI_LINE_NUM:= Sensor_DALI_LINE_NUM, 
 	//bCancelHoldTimerOccupancy:= bCancelHoldTimerOccupancy, 
	stSensorSetup := stDaliSensorSetup,
	arrInitErr=> arrInitErr, 
	arrInitDone=> arrInitDone,
	stPirSensorData:= stPirSensorData, 
	arrSensorScales:= arrSensorScales);*)
END_ACTION

END_PROGRAM

// ---- POUs/Alle_Rum/Rum_Med_DALI_Pir/Rum_1_218/P_Rum_1_218.TcPOU
PROGRAM P_Rum_1_218
VAR
(*
Rummet består af en lysgruppe og et ekstra armatur - L1G9 og L4S29 - på to forskellige linjer
Både gruppen og ekstra armatur afhænger af samme PIR-input - pir-adr. 7 - på DALI-linje 2.
Derfor oprettes to adskilte reguleringer med samme PV. Dvs., at knapfunktion og pirfunktion forbliver den samme.
*)

	arrfbLysGruppe			: ARRAY [1..2] OF FB_Light_Type_A;
	arrstDaliSetupGruppe	: ARRAY [1..2] OF SH_Light.ST_DALI_RoomSetup :=
	
													[(	byShrtAdr_Prim	:= 34, 
														byGrpAdr_Prim		:= 9, 
														eMod_Prim			:= E_DALIAddressType.Group, 
														//byShrtAdr_Sec		:= 1, 
														//byGrpAdr_Sec		:= 1, 
														//eMod_Sec			:= E_DALIAddressType.Short, 
														//byShrtAdr_Supl		:= 1,
														//byGrpAdr_Supl		:= 1,
														//eMod_Supl			:=  E_DALIAddressType.Short, 
														DALI_LINE_NUM_PRIM := arrDALI_LINE_NUM_LIGHT[1], 
														DALI_LINE_NUM_SEC := 0, //0 = ingen zonestyring/vinduerække
														DALI_LINE_NUM_SUPL := arrDALI_LINE_NUM_PENDANTS[1]),
														
													(	byShrtAdr_Prim	:= 29, 
														//byGrpAdr_Prim		:= 1, 
														eMod_Prim			:= E_DALIAddressType.Short, 
														//byShrtAdr_Sec		:= 1, 
														//byGrpAdr_Sec		:= 1, 
														//eMod_Sec			:= E_DALIAddressType.Short, 
														//byShrtAdr_Supl		:= 1,
														//byGrpAdr_Supl		:= 1,
														//eMod_Supl			:=  E_DALIAddressType.Short,
														DALI_LINE_NUM_PRIM := arrDALI_LINE_NUM_LIGHT[2], 
														DALI_LINE_NUM_SEC := 0, 
														DALI_LINE_NUM_SUPL := arrDALI_LINE_NUM_PENDANTS[2])];
														
	arrstLiveDataGruppe			: ARRAY [1..2] OF SH_Light.ST_LiveData;
	arrRunTuningGruppe			: ARRAY[1..2] OF BOOL;
	
	bTopButtonZone1				: BOOL;
	bTopButtonZone1_Visu		: BOOL;
	bBottomButtonZone1			: BOOL;
	bBottomButtonZone1_Visu	: BOOL;
	bButtonZone2					: BOOL;
	bNeighborRoomsPir			: BOOL;
	fLuxOn								: REAL;
	fLuxDim							: REAL;
	tPIRDim							: TIME;
	tPIROff							: TIME;
	fOffsetSec						: REAL := 20;
	bOccupiedRoom				: BOOL;

	bRunTuning						: BOOL;


// Sensor Settings
	fbSensor						: SH_Light.FB_NIKO_P46xx_1Pcs;
	//fbSensor					: SH_Light.FB_NIKO_P46xx_3Pcs;
	bySensorAddr				: BYTE := 7;
	//arrSensorAddr			: ARRAY[1..3] OF BYTE := [7,8,9];
	bInitialize						: BOOL := TRUE;
	stDaliSensorSetup			: ST_DALI_NIKOP46SetupData := (
																nSensitivityPIRSegmentA:=nSensitivityOccupancy,
																nSensitivityPIRSegmentB:=nSensitivityOccupancy,
																nSensitivityPIRSegmentC:=nSensitivityOccupancy);
	bInitErr							: BOOL;
	bInitDone						: BOOL;
	//arrInitErr					: ARRAY [1..3] OF BOOL;
	//arrInitDone				: ARRAY [1..3] OF BOOL;
	arrSensorScales				: ARRAY [1..10] OF SH_Light.ST_DALI_SensorScaleMode :=
																							[	(fMeassureMaxSensor := rMeassure_Zone4, fReadMaxSensor := rRead_Zone4),																						
																								9(())];
																								
	bCancelHoldTimerOccupancy	: BOOL;
(*	eEventPriorityOccupancy		: E_DALIEventPriority := E_DALIEVENTPRIORITY.Middle;
	nHoldTimerOccupancy			: WORD := 5; // Value in s. 	
	nReportTimerOccupancy		: BYTE := 120; // Value in s, Preset manufacturer value
	nDeadtimeTimerOccupancy		: WORD := 100; // Value in ms, Predefined Value of DALI Standard
	bCancelHoldTimerOccupancy	: BOOL; *)
	

(*	bEnableLuxEvent				: BOOL;
	eEventPriorityBrightness	: E_DALIEventPriority := E_DALIEVENTPRIORITY.Middle;
	nDeadtimeTimerBrightness	: WORD := 1500; // Value in ms, Predefined Value of DALI Standard
	nHysteresisBrightness		: BYTE := 2; // Value in %
	nHysteresisMinBrightness	: BYTE := 10; // Absolute Value, depending on the manufacturer specific resolution
	nReportTimerBrightness		: BYTE := 120; // Value in s, Preset manufacturer value
*)

	

//ModbusComm setup
	
	fbWriteSPLuxLevel			: SH_Light.FB_TwoVal_SelectOne_RTrigChange;
	fbWritePirDelayTIme		: SH_Light.FB_TwoVal_SelectOne_RTrigChange;
	stRoomDataPLC				: SH_Light.ST_RoomDataPLC	:=	(
																	uiPirOffDelayTime	:= 30,
																	uiSpLuxLevel			:= 500,
																	uiPirDimDelayTime	:= 15,
																	uiSpDimLuxLevel		:= 200);

	fbBallastOnHours			: SH_Light.FB_CountOnHours;
	bEnableHourCount		: BOOL := TRUE;
	
	//Non-persistent modbus data
	bPirActive_MB					AT%MX64.0	: BOOL;				//bPirLys i gammel kode
	uiActLuxLevel_MB			AT%MB68		: UINT;				//intHMIAktueltLux i gammel kode
	uiActLightLevelPct_MB	AT%MB72		: UINT;				//intDALI_Gruppe1_Lysniveau i gammel kode
	
	//For Conversion
	uiPirOffMinutes						: UINT;
	udTimeScaling						: UDINT := 60000;
	uiLuxOn								: UINT;
	
	//max values checks
	uiMaxLuxLevel						: UINT := 1023;
	uiMaxPirOffMinutes				: UINT := 180;


END_VAR

VAR CONSTANT
	Sensor_DALI_LINE_NUM				: BYTE := 2;
	arrDALI_LINE_NUM_LIGHT			: ARRAY[1..2] OF BYTE := [1,4]; //korrekt rækkefølge nødvendig
	arrDALI_LINE_NUM_PENDANTS: ARRAY[1..2] OF BYTE := [0,0]; //korrekt rækkefølge nødvendig. 0 = ingen pendler
	nSensitivityOccupancy						: BYTE:= 4; //setting Sensivity (0..4) 0 (Off), 1 (Min), 2(Low), 3(High) and 4 (Max)
END_VAR

VAR PERSISTENT
	stPirSensorData: SH_Light.ST_DALI_Sensor;
	arrstTuneDataGruppe: ARRAY [1..2] OF SH_Light.ST_TuneData_EX;
	
	uiPirOffDelayTime_MB		AT%MB66	    : UINT;				//intHMI_Pir_SetValue i gammel kode
	uiSPLuxLevel_MB			AT%MB70	    : UINT;				//intHMI_Lux_SetValue i gammel kode
	uiBallastOnHours_MB		AT%MB74		: UINT;				//dintHMILysbraendtimer1 i gammel kode
   	byOnHoursOverflowCount							: BYTE;
END_VAR

A_Buttons();
A_LightCtrl();
A_Sensor();
A_modbuscomm();

ACTION A_Buttons:
bTopButtonZone1		:= GVL_EnOcean.strEnOceanSwitch_Rum_1_218.bT2_ON OR bTopButtonZone1_Visu;
bBottomButtonZone1	:= GVL_EnOcean.strEnOceanSwitch_Rum_1_218.bT2_OFF OR bBottomButtonZone1_Visu;
END_ACTION

ACTION A_LightCtrl:

arrfbLysGruppe[1]( 
	nZoneID:= 1, 
	bButtonZone1:= bTopButtonZone1,
	bBottomButtonZone1 := bBottomButtonZone1, 
	//bButtonZone2:= bButtonZone2,
	fLuxOn:= fLuxOn, 
	fLuxDim:= fLuxDim, 
	tPIRDim:= tPIRDim, 
	tPIROff:= tPIROff, 
	fOffsetSec:= fOffsetSec, 
	bReInit:= , 
	stDaliSetup:= arrstDaliSetupGruppe[1], 
	ipCommunication_Prim:= P_DALI_Background.arrfbKL6821Communication[arrDALI_LINE_NUM_LIGHT[1]], 
	//ipCommunication_Sec:= P_DALI_Background.arrfbKL6821Communication[arrDALI_LINE_NUM_LIGHT[1]],
	//ipCommunication_Supl:= P_DALI_Background.arrfbKL6821Communication[arrDALI_LINE_NUM_PENDANTS[1]],
	fMinOutputPowerLevelRoom:= 15, 
	fMaxOutputPowerLevelRoom:= 100, 
	nCycleTimeInMS:= SH_Light.DALI_Param.nPlcTaskCycleTimeInMS*SH_Light.DALI_Param.nDimCmdCycleTimeFactor, 
	bRunTuning:= arrRunTuningGruppe[1], 
	bOccupiedRoom=> , 
	bError_Prim=> , 
	nError_Prim=> , 
	stTuneData:=arrstTuneDataGruppe[1] , 
	stPirSensorData:= stPirSensorData, 					//samme sensordata
	stLiveData:= arrstLiveDataGruppe[1]);


arrfbLysGruppe[2]( 
	nZoneID:= 1, 
	bButtonZone1:= bTopButtonZone1,
	bBottomButtonZone1 := bBottomButtonZone1, 
	bButtonZone2:= bButtonZone2,
	fLuxOn:= fLuxOn, 
	fLuxDim:= fLuxDim, 
	tPIRDim:= tPIRDim, 
	tPIROff:= tPIROff, 
	fOffsetSec:= fOffsetSec, 
	bReInit:= , 
	stDaliSetup:= arrstDaliSetupGruppe[2], 
	ipCommunication_Prim:= P_DALI_Background.arrfbKL6821Communication[arrDALI_LINE_NUM_LIGHT[2]], 
	//ipCommunication_Sec:= P_DALI_Background.arrfbKL6821Communication[arrDALI_LINE_NUM_LIGHT[2]],
	//ipCommunication_Supl:= P_DALI_Background.arrfbKL6821Communication[arrDALI_LINE_NUM_PENDANTS[2]],
	fMinOutputPowerLevelRoom:= 15, 
	fMaxOutputPowerLevelRoom:= 100, 
	nCycleTimeInMS:= SH_Light.DALI_Param.nPlcTaskCycleTimeInMS*SH_Light.DALI_Param.nDimCmdCycleTimeFactor, 
	bRunTuning:= arrRunTuningGruppe[2], 
	bOccupiedRoom=> , 
	bError_Prim=> , 
	nError_Prim=> , 
	stTuneData:=arrstTuneDataGruppe[2] , 
	stPirSensorData:= stPirSensorData, 					//samme sensordata
	stLiveData:= arrstLiveDataGruppe[2]);
END_ACTION

ACTION A_ModbusComm:
//Manage data for modbus communication

//Manage data for read-only in PLC
stRoomDataPLC.bPirActive			:= stPirSensorData.bPrc;
stRoomDataPLC.uiActLuxLevel			:= TO_UINT(TRUNC(stPirSensorData.fBrightness));
stRoomDataPLC.uiActLightLevelPct	:= TO_UINT(TRUNC(arrfbLysGruppe[1].fbBallast.fActlLgtLvl_Prim));
		//stRoomDataPLC.uiActLightLevelPct	:= TO_UINT(TRUNC(fbLys.fbBallast.fActlLgtLvl_Prim)); //if only one group light control
stRoomDataPLC.uiBallastOnHours		:= uiBallastOnHours_MB; //The calculation for BallastOnHours is stored directly to the MB register below


//Assign data for read-only to MB registers
bPirActive_MB			:= stRoomDataPLC.bPirActive;
uiActLuxLevel_MB		:= stRoomDataPLC.uiActLuxLevel;
uiActLightLevelPct_MB	:= stRoomDataPLC.uiActLightLevelPct;

	//calculate BallastOnHours
	fbBallastOnHours(
		bEnableHourCount	:= bEnableHourCount,
		bPauseCount			:= arrfbLysGruppe[1].fbLightCtrl.bOffZone1,
		uiOnHours			:= uiBallastOnHours_MB,			//OnHours is updated here
		byOverflowCount		:= byOnHoursOverflowCount);


//Manage data for read/write for both PLC and MB registers
fbWriteSPLuxLevel(	nMaxValOut	:= uiMaxLuxLevel,
					nValIn1		:= uiSPLuxLevel_MB,		//nValIn1 takes priotity in case of download or restart
					nValIn2		:= stRoomDataPLC.uiSpLuxLevel,
					nValOut		=> uiLuxOn
				);


fbWritePirDelayTIme(	nMaxValOut	:= uiMaxPirOffMinutes,
						nValIn1		:= uiPirOffDelayTime_MB,		//nValIn1 takes priotity in case of download or restart
						nValIn2		:= stRoomDataPLC.uiPirOffDelayTime,
						nValOut		=> uiPirOffMinutes
					);
					

//Convert read/write modbus data to appropriate datatypes in PLC
fLuxOn	:= TO_REAL(uiLuxOn);			
tPIROff	:= TO_TIME(uiPirOffMinutes*udTimeScaling); //Time conversion defaults to ms

fLuxDim	:= TO_REAL(stRoomDataPLC.uiSpDimLuxLevel);			
tPIRDim	:= TO_TIME(stRoomDataPLC.uiPirDimDelayTime*udTimeScaling); //Time conversion defaults to ms
END_ACTION

ACTION A_Sensor:

fbSensor.ipCommunication := P_DALI_Background.arrfbKL6821Communication[Sensor_DALI_LINE_NUM];

//only 1 sensor
fbSensor(
	byShrtAdr:= bySensorAddr,
	bInitialize:= bInitialize, 
	DALI_LINE_NUM:= Sensor_DALI_LINE_NUM, 
 	//bCancelHoldTimerOccupancy:= bCancelHoldTimerOccupancy, 
	stSensorSetup := stDaliSensorSetup,
	bInitErr=> bInitErr, 
	bInitDone=> bInitDone,
	stPirSensorData:= stPirSensorData, 
	arrSensorScales:= arrSensorScales);
	
(*//
//several sensors	
fbSensor(
	arrShrtAdr:= arrSensorAddr,
	bInitialize:= bInitialize, 
	DALI_LINE_NUM:= Sensor_DALI_LINE_NUM, 
 	//bCancelHoldTimerOccupancy:= bCancelHoldTimerOccupancy, 
	stSensorSetup := stDaliSensorSetup,
	arrInitErr=> arrInitErr, 
	arrInitDone=> arrInitDone,
	stPirSensorData:= stPirSensorData, 
	arrSensorScales:= arrSensorScales);*)
END_ACTION

END_PROGRAM

// ---- POUs/Alle_Rum/Rum_Med_DALI_Pir/Rum_1_219/P_Rum_1_219.TcPOU
PROGRAM P_Rum_1_219
VAR
(*
Rummet består af to lysgrupper - L1G5 og L4G4 - på to forskellige linjer
Begge grupper afhænger af samme PIR-input - pir-adr. 2 - på DALI-linje 4.
Derfor oprettes to adskilte reguleringer med samme PV. Dvs., at knapfunktion og pirfunktion forbliver den samme.
*)

	arrfbLysGruppe			: ARRAY [1..2] OF FB_Light_Type_A;
	arrstDaliSetupGruppe	: ARRAY [1..2] OF SH_Light.ST_DALI_RoomSetup :=
	
													[(	byShrtAdr_Prim	:= 24, 
														byGrpAdr_Prim		:= 5, 
														eMod_Prim			:= E_DALIAddressType.Group, 
														//byShrtAdr_Sec		:= 1, 
														//byGrpAdr_Sec		:= 1, 
														//eMod_Sec			:= E_DALIAddressType.Short, 
														//byShrtAdr_Supl		:= 1,
														//byGrpAdr_Supl		:= 1,
														//eMod_Supl			:=  E_DALIAddressType.Short, 
														DALI_LINE_NUM_PRIM := arrDALI_LINE_NUM_LIGHT[1], 
														DALI_LINE_NUM_SEC := 0, //0 = ingen zonestyring/vinduerække
														DALI_LINE_NUM_SUPL := arrDALI_LINE_NUM_PENDANTS[1]),
														
													(	byShrtAdr_Prim	:= 23, 
														byGrpAdr_Prim		:= 4, 
														eMod_Prim			:= E_DALIAddressType.Group, 
														//byShrtAdr_Sec		:= 1, 
														//byGrpAdr_Sec		:= 1, 
														//eMod_Sec			:= E_DALIAddressType.Short, 
														//byShrtAdr_Supl		:= 1,
														//byGrpAdr_Supl		:= 1,
														//eMod_Supl			:=  E_DALIAddressType.Short,
														DALI_LINE_NUM_PRIM := arrDALI_LINE_NUM_LIGHT[2], 
														DALI_LINE_NUM_SEC := 0, 
														DALI_LINE_NUM_SUPL := arrDALI_LINE_NUM_PENDANTS[2])];
														
	arrstLiveDataGruppe			: ARRAY [1..2] OF SH_Light.ST_LiveData;
	arrRunTuningGruppe			: ARRAY[1..2] OF BOOL;
	
	bTopButtonZone1				: BOOL;
	bTopButtonZone1_Visu		: BOOL;
	bBottomButtonZone1			: BOOL;
	bBottomButtonZone1_Visu	: BOOL;
	bButtonZone2					: BOOL;
	bNeighborRoomsPir			: BOOL;
	fLuxOn								: REAL;
	fLuxDim							: REAL;
	tPIRDim							: TIME;
	tPIROff							: TIME;
	fOffsetSec						: REAL := 20;
	bOccupiedRoom				: BOOL;

	bRunTuning						: BOOL;


// Sensor Settings
	fbSensor						: SH_Light.FB_NIKO_P46xx_1Pcs;
	//fbSensor					: SH_Light.FB_NIKO_P46xx_3Pcs;
	bySensorAddr				: BYTE := 2;
	//arrSensorAddr			: ARRAY[1..3] OF BYTE := [7,8,9];
	bInitialize						: BOOL := TRUE;
	stDaliSensorSetup			: ST_DALI_NIKOP46SetupData := (
																nSensitivityPIRSegmentA:=nSensitivityOccupancy,
																nSensitivityPIRSegmentB:=nSensitivityOccupancy,
																nSensitivityPIRSegmentC:=nSensitivityOccupancy);
	bInitErr							: BOOL;
	bInitDone						: BOOL;
	//arrInitErr					: ARRAY [1..3] OF BOOL;
	//arrInitDone				: ARRAY [1..3] OF BOOL;
	arrSensorScales				: ARRAY [1..10] OF SH_Light.ST_DALI_SensorScaleMode :=
																							[	(fMeassureMaxSensor := rMeassure_Zone3, fReadMaxSensor := rRead_Zone3),																							
																								9(())];
																								
	bCancelHoldTimerOccupancy	: BOOL;
(*	eEventPriorityOccupancy		: E_DALIEventPriority := E_DALIEVENTPRIORITY.Middle;
	nHoldTimerOccupancy			: WORD := 5; // Value in s. 	
	nReportTimerOccupancy		: BYTE := 120; // Value in s, Preset manufacturer value
	nDeadtimeTimerOccupancy		: WORD := 100; // Value in ms, Predefined Value of DALI Standard
	bCancelHoldTimerOccupancy	: BOOL; *)
	

(*	bEnableLuxEvent				: BOOL;
	eEventPriorityBrightness	: E_DALIEventPriority := E_DALIEVENTPRIORITY.Middle;
	nDeadtimeTimerBrightness	: WORD := 1500; // Value in ms, Predefined Value of DALI Standard
	nHysteresisBrightness		: BYTE := 2; // Value in %
	nHysteresisMinBrightness	: BYTE := 10; // Absolute Value, depending on the manufacturer specific resolution
	nReportTimerBrightness		: BYTE := 120; // Value in s, Preset manufacturer value
*)

	

//ModbusComm setup
	
	fbWriteSPLuxLevel			: SH_Light.FB_TwoVal_SelectOne_RTrigChange;
	fbWritePirDelayTIme		: SH_Light.FB_TwoVal_SelectOne_RTrigChange;
	stRoomDataPLC				: SH_Light.ST_RoomDataPLC	:=	(
																	uiPirOffDelayTime	:= 30,
																	uiSpLuxLevel			:= 500,
																	uiPirDimDelayTime	:= 15,
																	uiSpDimLuxLevel		:= 200);

	fbBallastOnHours			: SH_Light.FB_CountOnHours;
	bEnableHourCount		: BOOL := TRUE;
	
	//Non-persistent modbus data
	bPirActive_MB					AT%MX80.0	: BOOL;				//bPirLys i gammel kode
	uiActLuxLevel_MB			AT%MB84		: UINT;				//intHMIAktueltLux i gammel kode
	uiActLightLevelPct_MB	AT%MB88		: UINT;				//intDALI_Gruppe1_Lysniveau i gammel kode
	
	//For Conversion
	uiPirOffMinutes						: UINT;
	udTimeScaling						: UDINT := 60000;
	uiLuxOn								: UINT;
	
	//max values checks
	uiMaxLuxLevel						: UINT := 1023;
	uiMaxPirOffMinutes				: UINT := 180;


END_VAR

VAR CONSTANT
	Sensor_DALI_LINE_NUM				: BYTE := 4;
	arrDALI_LINE_NUM_LIGHT			: ARRAY[1..2] OF BYTE := [1,4]; //korrekt rækkefølge nødvendig
	arrDALI_LINE_NUM_PENDANTS: ARRAY[1..2] OF BYTE := [0,0]; //korrekt rækkefølge nødvendig. 0 = ingen pendler
	nSensitivityOccupancy						: BYTE:= 4; //setting Sensivity (0..4) 0 (Off), 1 (Min), 2(Low), 3(High) and 4 (Max)
END_VAR

VAR PERSISTENT
	stPirSensorData: SH_Light.ST_DALI_Sensor;
	arrstTuneDataGruppe: ARRAY [1..2] OF SH_Light.ST_TuneData_EX;
	
	uiPirOffDelayTime_MB		AT%MB82	    : UINT;				//intHMI_Pir_SetValue i gammel kode
	uiSPLuxLevel_MB			AT%MB86	    : UINT;				//intHMI_Lux_SetValue i gammel kode
	uiBallastOnHours_MB		AT%MB90		: UINT;				//dintHMILysbraendtimer1 i gammel kode
   	byOnHoursOverflowCount							: BYTE;
END_VAR

A_Buttons();
A_LightCtrl();
A_Sensor();
A_modbuscomm();

ACTION A_Buttons:
bTopButtonZone1		:= GVL_EnOcean.strEnOceanSwitch_Rum_1_219.bT1_ON OR bTopButtonZone1_Visu;
bBottomButtonZone1	:= GVL_EnOcean.strEnOceanSwitch_Rum_1_219.bT1_OFF OR bBottomButtonZone1_Visu;
END_ACTION

ACTION A_LightCtrl:

